(* IEC 61131-3 sources: TIA2AX/tests/V18/test_projects/expected/HW_2200330/ST30_PLC, 7 files *)

(* ---- HwIdentifiers.st ---- *)
TYPE
	HwIdentifiers : WORD
	(
		ST30_PLC_Profilschiene_0 :=	WORD#256,
		ST30_PLC :=	WORD#48,
		ST30_PLC_Card_reader_writer_1 :=	WORD#51,
		ST30_PLC_CPU_display_1 :=	WORD#54,
		ST30_PLC_OPC_UA_1 :=	WORD#117,
		ST30_PLC_DP_interface_1 :=	WORD#60,
		ST30_PLC_PROFINET_interface_1 :=	WORD#64,
		ST30_PLC_PROFINET_interface_1_Port_1 :=	WORD#65,
		ST30_PLC_PROFINET_interface_1_Port_2 :=	WORD#66,
		ST30_PLC_PROFINET_interface_2 :=	WORD#72,
		ST30_PLC_PROFINET_interface_2_Port_1 :=	WORD#73,
		ST30_Switch_SCALANCE_X_rack :=	WORD#436,
		ST30_Switch :=	WORD#437,
		ST30_Switch_ST30_Switch :=	WORD#438,
		ST30_Switch_SCALANCE_interface_1 :=	WORD#439,
		ST30_Switch_SCALANCE_interface_1_Port_1 :=	WORD#440,
		ST30_Switch_SCALANCE_interface_1_Port_2 :=	WORD#441,
		ST30_Switch_SCALANCE_interface_1_Port_3 :=	WORD#442,
		ST30_Switch_SCALANCE_interface_1_Port_4 :=	WORD#443,
		ST30_Switch_SCALANCE_interface_1_Port_5 :=	WORD#444,
		ST30_Switch_SCALANCE_interface_1_Port_6 :=	WORD#445,
		ST30_Switch_SCALANCE_interface_1_Port_7 :=	WORD#446,
		ST30_Switch_SCALANCE_interface_1_Port_8 :=	WORD#447,
		ST30_ET200SP_Rack_0 :=	WORD#276,
		ST30_ET200SP :=	WORD#277,
		ST30_ET200SP_ST30_ET200SP :=	WORD#258,
		ST30_ET200SP_PROFINET_interface :=	WORD#259,
		ST30_ET200SP_PROFINET_interface_Port_1 :=	WORD#260,
		ST30_ET200SP_PROFINET_interface_Port_2 :=	WORD#261,
		ST30_ET200SP_BA_2xRJ45 :=	WORD#260,
		ST30_ET200SP_CM_4xIO_Link_1 :=	WORD#262,
		ST30_ET200SP_CM_4xIO_Link_2 :=	WORD#263,
		ST30_ET200SP_DI_16x24VDC_ST_1 :=	WORD#264,
		ST30_ET200SP_DI_16x24VDC_ST_2 :=	WORD#265,
		ST30_ET200SP_DI_16x24VDC_ST_3 :=	WORD#266,
		ST30_ET200SP_DI_16x24VDC_ST_4 :=	WORD#267,
		ST30_ET200SP_DI_16x24VDC_ST_5 :=	WORD#268,
		ST30_ET200SP_DI_16x24VDC_ST_6 :=	WORD#269,
		ST30_ET200SP_DQ_16x24VDC_0_5A_ST_1 :=	WORD#270,
		ST30_ET200SP_DQ_16x24VDC_0_5A_ST_2 :=	WORD#271,
		ST30_ET200SP_DQ_16x24VDC_0_5A_ST_3 :=	WORD#272,
		ST30_ET200SP_DQ_16x24VDC_0_5A_ST_4 :=	WORD#273,
		ST30_ET200SP_Servermodul_1 :=	WORD#274,
		ST30_CPX_PN_IO_Interface :=	WORD#281,
		ST30_CPX_PN_IO_Interface_Port_1 :=	WORD#282,
		ST30_CPX_PN_IO_Interface_Port_2 :=	WORD#283,
		ST30_CPX_CPX :=	WORD#284,
		ST30_CPX_MPA1S_VMPA1_FB_EMS_8_8DO_1 :=	WORD#285,
		ST30_CPX_MPA1G_VMPA1_FB_EMG_8_8DO_1 :=	WORD#286,
		ST30_CPX_MPA1G_VMPA1_FB_EMG_8_8DO_2 :=	WORD#287,
		ST30_1_ACT350_Rack :=	WORD#289,
		ST30_1_ACT350 :=	WORD#290,
		ST30_1_ACT350_PROFINET :=	WORD#291,
		ST30_1_ACT350_PROFINET_Port_1 :=	WORD#292,
		ST30_1_ACT350_PROFINET_Port_2 :=	WORD#293,
		ST30_1_ACT350_DAP_2_Block_Parameter :=	WORD#294,
		ST30_1_ACT350_Measuring_Block_1 :=	WORD#295,
		ST30_1_ACT350_Measuring_Block_1_Parameter_Access_Point :=	WORD#296,
		ST30_1_ACT350_Measuring_Block_1_MB_Command_Value :=	WORD#297,
		ST30_1_ACT350_Measuring_Block_1_MB_Channel_Mask :=	WORD#298,
		ST30_1_ACT350_Measuring_Block_1_MB_Command :=	WORD#299,
		ST30_1_ACT350_Measuring_Block_1_MB_Measuring_Value :=	WORD#300,
		ST30_1_ACT350_Measuring_Block_1_MB_Device_Status :=	WORD#301,
		ST30_1_ACT350_Measuring_Block_1_MB_Response :=	WORD#302,
		ST30_1_ACT350_Status_Block_1 :=	WORD#303,
		ST30_1_ACT350_Status_Block_1_Parameter_Access_Point :=	WORD#304,
		ST30_1_ACT350_Status_Block_1_SB_Reserved_1 :=	WORD#305,
		ST30_1_ACT350_Status_Block_1_SB_Reserved_2 :=	WORD#306,
		ST30_1_ACT350_Status_Block_1_SB_Reserved_3 :=	WORD#307,
		ST30_1_ACT350_Status_Block_1_SB_Command :=	WORD#308,
		ST30_1_ACT350_Status_Block_1_SB_Status_Group_1 :=	WORD#309,
		ST30_1_ACT350_Status_Block_1_SB_Status_Group_2 :=	WORD#310,
		ST30_1_ACT350_Status_Block_1_SB_Status_Group_3 :=	WORD#311,
		ST30_1_ACT350_Status_Block_1_SB_Response :=	WORD#312,
		ST30_1_DM260_Rack :=	WORD#314,
		ST30_1_DM260 :=	WORD#315,
		ST30_1_DM260_Interface :=	WORD#316,
		ST30_1_DM260_Interface_Port_1 :=	WORD#317,
		ST30_1_DM260_DataMan_260 :=	WORD#318,
		ST30_1_DM260_Acquisition_Control_1 :=	WORD#319,
		ST30_1_DM260_Acquisition_Status_1 :=	WORD#320,
		ST30_1_DM260_Results_Control_1 :=	WORD#321,
		ST30_1_DM260_Results_Status_1 :=	WORD#322,
		ST30_1_DM260_Soft_Event_Control_1 :=	WORD#323,
		ST30_1_DM260_User_Data_64_bytes_1 :=	WORD#324,
		ST30_1_DM260_Result_Data_64_bytes_1 :=	WORD#325,
		ST30_1_CMMT_AS_X_PN_IO_Interface :=	WORD#329,
		ST30_1_CMMT_AS_X_PN_IO_Interface_Port_1 :=	WORD#330,
		ST30_1_CMMT_AS_X_PN_IO_Interface_Port_2 :=	WORD#331,
		ST30_1_CMMT_AS_X_CMMT_AS_V1 :=	WORD#332,
		ST30_1_CMMT_AS_X_DO_SERVO_1_Module_Access_Point :=	WORD#334,
		ST30_1_CMMT_AS_X_DO_SERVO_1_Siemens_telegram_111_PZD_12_12 :=	WORD#335,
		ST30_1_CMMT_AS_X_Siemens_telegram_111_PZD_12_12 :=	WORD#335,
		ST30_1_CMMT_AS_Y_PN_IO_Interface :=	WORD#339,
		ST30_1_CMMT_AS_Y_PN_IO_Interface_Port_1 :=	WORD#340,
		ST30_1_CMMT_AS_Y_PN_IO_Interface_Port_2 :=	WORD#341,
		ST30_1_CMMT_AS_Y_CMMT_AS_V1 :=	WORD#342,
		ST30_1_CMMT_AS_Y_DO_SERVO_1_Module_Access_Point :=	WORD#344,
		ST30_1_CMMT_AS_Y_DO_SERVO_1_Siemens_telegram_111_PZD_12_12 :=	WORD#345,
		ST30_1_CMMT_AS_Y_Siemens_telegram_111_PZD_12_12 :=	WORD#345,
		ST30_1_CMMT_AS_Z_PN_IO_Interface :=	WORD#349,
		ST30_1_CMMT_AS_Z_PN_IO_Interface_Port_1 :=	WORD#350,
		ST30_1_CMMT_AS_Z_PN_IO_Interface_Port_2 :=	WORD#351,
		ST30_1_CMMT_AS_Z_CMMT_AS_V1 :=	WORD#352,
		ST30_1_CMMT_AS_Z_DO_SERVO_1_Module_Access_Point :=	WORD#354,
		ST30_1_CMMT_AS_Z_DO_SERVO_1_Siemens_telegram_111_PZD_12_12 :=	WORD#355,
		ST30_1_CMMT_AS_Z_Siemens_telegram_111_PZD_12_12 :=	WORD#355,
		ST30_HMI_ConnectionBox_Connection_Box :=	WORD#357,
		ST30_HMI_ConnectionBox :=	WORD#358,
		ST30_HMI_ConnectionBox_ST30_HMI_ConnectionBox :=	WORD#359,
		ST30_HMI_ConnectionBox_SCALANCE_interface_1 :=	WORD#360,
		ST30_HMI_ConnectionBox_SCALANCE_interface_1_Port_1 :=	WORD#361,
		ST30_HMI_ConnectionBox_SCALANCE_interface_1_Port_2 :=	WORD#362,
		ST30_HMI_ConnectionBox_SCALANCE_interface_1_Port_3 :=	WORD#363,
		ST30_2_ACT350_Rack :=	WORD#365,
		ST30_2_ACT350 :=	WORD#366,
		ST30_2_ACT350_PROFINET :=	WORD#367,
		ST30_2_ACT350_PROFINET_Port_1 :=	WORD#368,
		ST30_2_ACT350_PROFINET_Port_2 :=	WORD#369,
		ST30_2_ACT350_DAP_2_Block_Parameter :=	WORD#370,
		ST30_2_ACT350_Measuring_Block_1 :=	WORD#371,
		ST30_2_ACT350_Measuring_Block_1_Parameter_Access_Point :=	WORD#372,
		ST30_2_ACT350_Measuring_Block_1_MB_Command_Value :=	WORD#373,
		ST30_2_ACT350_Measuring_Block_1_MB_Channel_Mask :=	WORD#374,
		ST30_2_ACT350_Measuring_Block_1_MB_Command :=	WORD#375,
		ST30_2_ACT350_Measuring_Block_1_MB_Measuring_Value :=	WORD#376,
		ST30_2_ACT350_Measuring_Block_1_MB_Device_Status :=	WORD#377,
		ST30_2_ACT350_Measuring_Block_1_MB_Response :=	WORD#378,
		ST30_2_ACT350_Status_Block_1 :=	WORD#379,
		ST30_2_ACT350_Status_Block_1_Parameter_Access_Point :=	WORD#380,
		ST30_2_ACT350_Status_Block_1_SB_Reserved_1 :=	WORD#381,
		ST30_2_ACT350_Status_Block_1_SB_Reserved_2 :=	WORD#382,
		ST30_2_ACT350_Status_Block_1_SB_Reserved_3 :=	WORD#383,
		ST30_2_ACT350_Status_Block_1_SB_Command :=	WORD#384,
		ST30_2_ACT350_Status_Block_1_SB_Status_Group_1 :=	WORD#385,
		ST30_2_ACT350_Status_Block_1_SB_Status_Group_2 :=	WORD#386,
		ST30_2_ACT350_Status_Block_1_SB_Status_Group_3 :=	WORD#387,
		ST30_2_ACT350_Status_Block_1_SB_Response :=	WORD#388,
		ST30_2_CMMT_AS_X_PN_IO_Interface :=	WORD#392,
		ST30_2_CMMT_AS_X_PN_IO_Interface_Port_1 :=	WORD#393,
		ST30_2_CMMT_AS_X_PN_IO_Interface_Port_2 :=	WORD#394,
		ST30_2_CMMT_AS_X_CMMT_AS_V1 :=	WORD#395,
		ST30_2_CMMT_AS_X_DO_SERVO_1_Module_Access_Point :=	WORD#397,
		ST30_2_CMMT_AS_X_DO_SERVO_1_Siemens_telegram_111_PZD_12_12 :=	WORD#398,
		ST30_2_CMMT_AS_X_Siemens_telegram_111_PZD_12_12 :=	WORD#398,
		ST30_2_CMMT_AS_Y_PN_IO_Interface :=	WORD#402,
		ST30_2_CMMT_AS_Y_PN_IO_Interface_Port_1 :=	WORD#403,
		ST30_2_CMMT_AS_Y_PN_IO_Interface_Port_2 :=	WORD#404,
		ST30_2_CMMT_AS_Y_CMMT_AS_V1 :=	WORD#405,
		ST30_2_CMMT_AS_Y_DO_SERVO_1_Module_Access_Point :=	WORD#407,
		ST30_2_CMMT_AS_Y_DO_SERVO_1_Siemens_telegram_111_PZD_12_12 :=	WORD#408,
		ST30_2_CMMT_AS_Y_Siemens_telegram_111_PZD_12_12 :=	WORD#408,
		ST30_2_CMMT_AS_Z_PN_IO_Interface :=	WORD#412,
		ST30_2_CMMT_AS_Z_PN_IO_Interface_Port_1 :=	WORD#413,
		ST30_2_CMMT_AS_Z_PN_IO_Interface_Port_2 :=	WORD#414,
		ST30_2_CMMT_AS_Z_CMMT_AS_V1 :=	WORD#415,
		ST30_2_CMMT_AS_Z_DO_SERVO_1_Module_Access_Point :=	WORD#417,
		ST30_2_CMMT_AS_Z_DO_SERVO_1_Siemens_telegram_111_PZD_12_12 :=	WORD#418,
		ST30_2_CMMT_AS_Z_Siemens_telegram_111_PZD_12_12 :=	WORD#418,
		ST30_2_DM260_Rack :=	WORD#420,
		ST30_2_DM260 :=	WORD#421,
		ST30_2_DM260_Interface :=	WORD#422,
		ST30_2_DM260_Interface_Port_1 :=	WORD#423,
		ST30_2_DM260_DataMan_260 :=	WORD#424,
		ST30_2_DM260_Acquisition_Control_1 :=	WORD#425,
		ST30_2_DM260_Acquisition_Status_1 :=	WORD#426,
		ST30_2_DM260_Results_Control_1 :=	WORD#427,
		ST30_2_DM260_Results_Status_1 :=	WORD#428,
		ST30_2_DM260_Soft_Event_Control_1 :=	WORD#429,
		ST30_2_DM260_User_Data_64_bytes_1 :=	WORD#430,
		ST30_2_DM260_Result_Data_64_bytes_1 :=	WORD#431,
		NONE:= WORD#0
	);
END_TYPE

(* ---- HwInputs.st ---- *)
TYPE
	HwInputs : STRUCT
		ST30_ET200SP_CM_4xIO_Link_1 AT %B100 : ARRAY[0..31] OF BYTE;
		ST30_ET200SP_CM_4xIO_Link_2 AT %B132 : ARRAY[0..31] OF BYTE;
		ST30_ET200SP_DI_16x24VDC_ST_1 AT %B0 : WORD;
		ST30_ET200SP_DI_16x24VDC_ST_2 AT %B2 : WORD;
		ST30_ET200SP_DI_16x24VDC_ST_3 AT %B4 : WORD;
		ST30_ET200SP_DI_16x24VDC_ST_4 AT %B6 : WORD;
		ST30_ET200SP_DI_16x24VDC_ST_5 AT %B8 : WORD;
		ST30_ET200SP_DI_16x24VDC_ST_6 AT %B10 : WORD;
		ST30_1_ACT350_Measuring_Block_1_MB_Measuring_Value AT %B1000 : DWORD;
		ST30_1_ACT350_Measuring_Block_1_MB_Device_Status AT %B1004 : WORD;
		ST30_1_ACT350_Measuring_Block_1_MB_Response AT %B1006 : WORD;
		ST30_1_ACT350_Status_Block_1_SB_Status_Group_1 AT %B1010 : WORD;
		ST30_1_ACT350_Status_Block_1_SB_Status_Group_2 AT %B1012 : WORD;
		ST30_1_ACT350_Status_Block_1_SB_Status_Group_3 AT %B1014 : WORD;
		ST30_1_ACT350_Status_Block_1_SB_Response AT %B1016 : WORD;
		ST30_1_DM260_Acquisition_Status_1 AT %B1500 : ARRAY[0..2] OF BYTE;
		ST30_1_DM260_Results_Status_1 AT %B1503 : BYTE;
		ST30_1_DM260_Soft_Event_Control_1 AT %B1504 : BYTE;
		ST30_1_DM260_Result_Data_64_bytes_1 AT %B1510 : ARRAY[0..71] OF BYTE;
		ST30_1_CMMT_AS_X_DO_SERVO_1_Siemens_telegram_111_PZD_12_12 AT %B1100 : ARRAY[0..23] OF BYTE;
		ST30_1_CMMT_AS_Y_DO_SERVO_1_Siemens_telegram_111_PZD_12_12 AT %B1200 : ARRAY[0..23] OF BYTE;
		ST30_1_CMMT_AS_Z_DO_SERVO_1_Siemens_telegram_111_PZD_12_12 AT %B1300 : ARRAY[0..23] OF BYTE;
		ST30_2_ACT350_Measuring_Block_1_MB_Measuring_Value AT %B2000 : DWORD;
		ST30_2_ACT350_Measuring_Block_1_MB_Device_Status AT %B2004 : WORD;
		ST30_2_ACT350_Measuring_Block_1_MB_Response AT %B2006 : WORD;
		ST30_2_ACT350_Status_Block_1_SB_Status_Group_1 AT %B2010 : WORD;
		ST30_2_ACT350_Status_Block_1_SB_Status_Group_2 AT %B2012 : WORD;
		ST30_2_ACT350_Status_Block_1_SB_Status_Group_3 AT %B2014 : WORD;
		ST30_2_ACT350_Status_Block_1_SB_Response AT %B2016 : WORD;
		ST30_2_CMMT_AS_X_DO_SERVO_1_Siemens_telegram_111_PZD_12_12 AT %B2100 : ARRAY[0..23] OF BYTE;
		ST30_2_CMMT_AS_Y_DO_SERVO_1_Siemens_telegram_111_PZD_12_12 AT %B2200 : ARRAY[0..23] OF BYTE;
		ST30_2_CMMT_AS_Z_DO_SERVO_1_Siemens_telegram_111_PZD_12_12 AT %B2300 : ARRAY[0..23] OF BYTE;
		ST30_2_DM260_Acquisition_Status_1 AT %B2500 : ARRAY[0..2] OF BYTE;
		ST30_2_DM260_Results_Status_1 AT %B2503 : BYTE;
		ST30_2_DM260_Soft_Event_Control_1 AT %B2504 : BYTE;
		ST30_2_DM260_Result_Data_64_bytes_1 AT %B2510 : ARRAY[0..71] OF BYTE;
	END_STRUCT;
END_TYPE

(* ---- HwOutputs.st ---- *)
TYPE
	HwOutputs : STRUCT
		ST30_ET200SP_CM_4xIO_Link_1 AT %B100 : ARRAY[0..31] OF BYTE;
		ST30_ET200SP_CM_4xIO_Link_2 AT %B132 : ARRAY[0..31] OF BYTE;
		ST30_ET200SP_DQ_16x24VDC_0_5A_ST_1 AT %B0 : WORD;
		ST30_ET200SP_DQ_16x24VDC_0_5A_ST_2 AT %B2 : WORD;
		ST30_ET200SP_DQ_16x24VDC_0_5A_ST_3 AT %B4 : WORD;
		ST30_ET200SP_DQ_16x24VDC_0_5A_ST_4 AT %B6 : WORD;
		ST30_CPX_MPA1S_VMPA1_FB_EMS_8_8DO_1 AT %B200 : BYTE;
		ST30_CPX_MPA1G_VMPA1_FB_EMG_8_8DO_1 AT %B201 : BYTE;
		ST30_CPX_MPA1G_VMPA1_FB_EMG_8_8DO_2 AT %B202 : BYTE;
		ST30_1_ACT350_Measuring_Block_1_MB_Command_Value AT %B1000 : DWORD;
		ST30_1_ACT350_Measuring_Block_1_MB_Channel_Mask AT %B1004 : WORD;
		ST30_1_ACT350_Measuring_Block_1_MB_Command AT %B1006 : WORD;
		ST30_1_ACT350_Status_Block_1_SB_Reserved_1 AT %B1010 : WORD;
		ST30_1_ACT350_Status_Block_1_SB_Reserved_2 AT %B1012 : WORD;
		ST30_1_ACT350_Status_Block_1_SB_Reserved_3 AT %B1014 : WORD;
		ST30_1_ACT350_Status_Block_1_SB_Command AT %B1016 : WORD;
		ST30_1_DM260_Acquisition_Control_1 AT %B1500 : BYTE;
		ST30_1_DM260_Results_Control_1 AT %B1503 : BYTE;
		ST30_1_DM260_Soft_Event_Control_1 AT %B1504 : BYTE;
		ST30_1_DM260_User_Data_64_bytes_1 AT %B1510 : ARRAY[0..67] OF BYTE;
		ST30_1_CMMT_AS_X_DO_SERVO_1_Siemens_telegram_111_PZD_12_12 AT %B1100 : ARRAY[0..23] OF BYTE;
		ST30_1_CMMT_AS_Y_DO_SERVO_1_Siemens_telegram_111_PZD_12_12 AT %B1200 : ARRAY[0..23] OF BYTE;
		ST30_1_CMMT_AS_Z_DO_SERVO_1_Siemens_telegram_111_PZD_12_12 AT %B1300 : ARRAY[0..23] OF BYTE;
		ST30_2_ACT350_Measuring_Block_1_MB_Command_Value AT %B2000 : DWORD;
		ST30_2_ACT350_Measuring_Block_1_MB_Channel_Mask AT %B2004 : WORD;
		ST30_2_ACT350_Measuring_Block_1_MB_Command AT %B2006 : WORD;
		ST30_2_ACT350_Status_Block_1_SB_Reserved_1 AT %B2010 : WORD;
		ST30_2_ACT350_Status_Block_1_SB_Reserved_2 AT %B2012 : WORD;
		ST30_2_ACT350_Status_Block_1_SB_Reserved_3 AT %B2014 : WORD;
		ST30_2_ACT350_Status_Block_1_SB_Command AT %B2016 : WORD;
		ST30_2_CMMT_AS_X_DO_SERVO_1_Siemens_telegram_111_PZD_12_12 AT %B2100 : ARRAY[0..23] OF BYTE;
		ST30_2_CMMT_AS_Y_DO_SERVO_1_Siemens_telegram_111_PZD_12_12 AT %B2200 : ARRAY[0..23] OF BYTE;
		ST30_2_CMMT_AS_Z_DO_SERVO_1_Siemens_telegram_111_PZD_12_12 AT %B2300 : ARRAY[0..23] OF BYTE;
		ST30_2_DM260_Acquisition_Control_1 AT %B2500 : BYTE;
		ST30_2_DM260_Results_Control_1 AT %B2503 : BYTE;
		ST30_2_DM260_Soft_Event_Control_1 AT %B2504 : BYTE;
		ST30_2_DM260_User_Data_64_bytes_1 AT %B2510 : ARRAY[0..67] OF BYTE;
	END_STRUCT;
END_TYPE

(* ---- PlcInputs.st ---- *)
TYPE
	PlcInputs : STRUCT
		ST30_ET200SP_CM_4xIO_Link_1 : ARRAY[0..31] OF BYTE;
		ST30_ET200SP_CM_4xIO_Link_2 : ARRAY[0..31] OF BYTE;
		ST30_ET200SP_DI_16x24VDC_ST_1 : WORD;
		ST30_ET200SP_DI_16x24VDC_ST_2 : WORD;
		ST30_ET200SP_DI_16x24VDC_ST_3 : WORD;
		ST30_ET200SP_DI_16x24VDC_ST_4 : WORD;
		ST30_ET200SP_DI_16x24VDC_ST_5 : WORD;
		ST30_ET200SP_DI_16x24VDC_ST_6 : WORD;
		ST30_1_ACT350_Measuring_Block_1_MB_Measuring_Value : DWORD;
		ST30_1_ACT350_Measuring_Block_1_MB_Device_Status : WORD;
		ST30_1_ACT350_Measuring_Block_1_MB_Response : WORD;
		ST30_1_ACT350_Status_Block_1_SB_Status_Group_1 : WORD;
		ST30_1_ACT350_Status_Block_1_SB_Status_Group_2 : WORD;
		ST30_1_ACT350_Status_Block_1_SB_Status_Group_3 : WORD;
		ST30_1_ACT350_Status_Block_1_SB_Response : WORD;
		ST30_1_DM260_Acquisition_Status_1 : ARRAY[0..2] OF BYTE;
		ST30_1_DM260_Results_Status_1 : BYTE;
		ST30_1_DM260_Soft_Event_Control_1 : BYTE;
		ST30_1_DM260_Result_Data_64_bytes_1 : ARRAY[0..71] OF BYTE;
		ST30_1_CMMT_AS_X_DO_SERVO_1_Siemens_telegram_111_PZD_12_12 : ARRAY[0..23] OF BYTE;
		ST30_1_CMMT_AS_Y_DO_SERVO_1_Siemens_telegram_111_PZD_12_12 : ARRAY[0..23] OF BYTE;
		ST30_1_CMMT_AS_Z_DO_SERVO_1_Siemens_telegram_111_PZD_12_12 : ARRAY[0..23] OF BYTE;
		ST30_2_ACT350_Measuring_Block_1_MB_Measuring_Value : DWORD;
		ST30_2_ACT350_Measuring_Block_1_MB_Device_Status : WORD;
		ST30_2_ACT350_Measuring_Block_1_MB_Response : WORD;
		ST30_2_ACT350_Status_Block_1_SB_Status_Group_1 : WORD;
		ST30_2_ACT350_Status_Block_1_SB_Status_Group_2 : WORD;
		ST30_2_ACT350_Status_Block_1_SB_Status_Group_3 : WORD;
		ST30_2_ACT350_Status_Block_1_SB_Response : WORD;
		ST30_2_CMMT_AS_X_DO_SERVO_1_Siemens_telegram_111_PZD_12_12 : ARRAY[0..23] OF BYTE;
		ST30_2_CMMT_AS_Y_DO_SERVO_1_Siemens_telegram_111_PZD_12_12 : ARRAY[0..23] OF BYTE;
		ST30_2_CMMT_AS_Z_DO_SERVO_1_Siemens_telegram_111_PZD_12_12 : ARRAY[0..23] OF BYTE;
		ST30_2_DM260_Acquisition_Status_1 : ARRAY[0..2] OF BYTE;
		ST30_2_DM260_Results_Status_1 : BYTE;
		ST30_2_DM260_Soft_Event_Control_1 : BYTE;
		ST30_2_DM260_Result_Data_64_bytes_1 : ARRAY[0..71] OF BYTE;
	END_STRUCT;
END_TYPE

(* ---- PlcOutputs.st ---- *)
TYPE
	PlcOutputs : STRUCT
		ST30_ET200SP_CM_4xIO_Link_1 : ARRAY[0..31] OF BYTE;
		ST30_ET200SP_CM_4xIO_Link_2 : ARRAY[0..31] OF BYTE;
		ST30_ET200SP_DQ_16x24VDC_0_5A_ST_1 : WORD;
		ST30_ET200SP_DQ_16x24VDC_0_5A_ST_2 : WORD;
		ST30_ET200SP_DQ_16x24VDC_0_5A_ST_3 : WORD;
		ST30_ET200SP_DQ_16x24VDC_0_5A_ST_4 : WORD;
		ST30_CPX_MPA1S_VMPA1_FB_EMS_8_8DO_1 : BYTE;
		ST30_CPX_MPA1G_VMPA1_FB_EMG_8_8DO_1 : BYTE;
		ST30_CPX_MPA1G_VMPA1_FB_EMG_8_8DO_2 : BYTE;
		ST30_1_ACT350_Measuring_Block_1_MB_Command_Value : DWORD;
		ST30_1_ACT350_Measuring_Block_1_MB_Channel_Mask : WORD;
		ST30_1_ACT350_Measuring_Block_1_MB_Command : WORD;
		ST30_1_ACT350_Status_Block_1_SB_Reserved_1 : WORD;
		ST30_1_ACT350_Status_Block_1_SB_Reserved_2 : WORD;
		ST30_1_ACT350_Status_Block_1_SB_Reserved_3 : WORD;
		ST30_1_ACT350_Status_Block_1_SB_Command : WORD;
		ST30_1_DM260_Acquisition_Control_1 : BYTE;
		ST30_1_DM260_Results_Control_1 : BYTE;
		ST30_1_DM260_Soft_Event_Control_1 : BYTE;
		ST30_1_DM260_User_Data_64_bytes_1 : ARRAY[0..67] OF BYTE;
		ST30_1_CMMT_AS_X_DO_SERVO_1_Siemens_telegram_111_PZD_12_12 : ARRAY[0..23] OF BYTE;
		ST30_1_CMMT_AS_Y_DO_SERVO_1_Siemens_telegram_111_PZD_12_12 : ARRAY[0..23] OF BYTE;
		ST30_1_CMMT_AS_Z_DO_SERVO_1_Siemens_telegram_111_PZD_12_12 : ARRAY[0..23] OF BYTE;
		ST30_2_ACT350_Measuring_Block_1_MB_Command_Value : DWORD;
		ST30_2_ACT350_Measuring_Block_1_MB_Channel_Mask : WORD;
		ST30_2_ACT350_Measuring_Block_1_MB_Command : WORD;
		ST30_2_ACT350_Status_Block_1_SB_Reserved_1 : WORD;
		ST30_2_ACT350_Status_Block_1_SB_Reserved_2 : WORD;
		ST30_2_ACT350_Status_Block_1_SB_Reserved_3 : WORD;
		ST30_2_ACT350_Status_Block_1_SB_Command : WORD;
		ST30_2_CMMT_AS_X_DO_SERVO_1_Siemens_telegram_111_PZD_12_12 : ARRAY[0..23] OF BYTE;
		ST30_2_CMMT_AS_Y_DO_SERVO_1_Siemens_telegram_111_PZD_12_12 : ARRAY[0..23] OF BYTE;
		ST30_2_CMMT_AS_Z_DO_SERVO_1_Siemens_telegram_111_PZD_12_12 : ARRAY[0..23] OF BYTE;
		ST30_2_DM260_Acquisition_Control_1 : BYTE;
		ST30_2_DM260_Results_Control_1 : BYTE;
		ST30_2_DM260_Soft_Event_Control_1 : BYTE;
		ST30_2_DM260_User_Data_64_bytes_1 : ARRAY[0..67] OF BYTE;
	END_STRUCT;
END_TYPE

(* ---- CopyInputs.st ---- *)
FUNCTION CopyInputs
	VAR_EXTERNAL
		HwInputs : HwInputs;
		PlcInputs : PlcInputs;
	END_VAR
	PlcInputs.ST30_ET200SP_CM_4xIO_Link_1[0] := HwInputs.ST30_ET200SP_CM_4xIO_Link_1[0];
	PlcInputs.ST30_ET200SP_CM_4xIO_Link_1[1] := HwInputs.ST30_ET200SP_CM_4xIO_Link_1[1];
	PlcInputs.ST30_ET200SP_CM_4xIO_Link_1[2] := HwInputs.ST30_ET200SP_CM_4xIO_Link_1[2];
	PlcInputs.ST30_ET200SP_CM_4xIO_Link_1[3] := HwInputs.ST30_ET200SP_CM_4xIO_Link_1[3];
	PlcInputs.ST30_ET200SP_CM_4xIO_Link_1[4] := HwInputs.ST30_ET200SP_CM_4xIO_Link_1[4];
	PlcInputs.ST30_ET200SP_CM_4xIO_Link_1[5] := HwInputs.ST30_ET200SP_CM_4xIO_Link_1[5];
	PlcInputs.ST30_ET200SP_CM_4xIO_Link_1[6] := HwInputs.ST30_ET200SP_CM_4xIO_Link_1[6];
	PlcInputs.ST30_ET200SP_CM_4xIO_Link_1[7] := HwInputs.ST30_ET200SP_CM_4xIO_Link_1[7];
	PlcInputs.ST30_ET200SP_CM_4xIO_Link_1[8] := HwInputs.ST30_ET200SP_CM_4xIO_Link_1[8];
	PlcInputs.ST30_ET200SP_CM_4xIO_Link_1[9] := HwInputs.ST30_ET200SP_CM_4xIO_Link_1[9];
	PlcInputs.ST30_ET200SP_CM_4xIO_Link_1[10] := HwInputs.ST30_ET200SP_CM_4xIO_Link_1[10];
	PlcInputs.ST30_ET200SP_CM_4xIO_Link_1[11] := HwInputs.ST30_ET200SP_CM_4xIO_Link_1[11];
	PlcInputs.ST30_ET200SP_CM_4xIO_Link_1[12] := HwInputs.ST30_ET200SP_CM_4xIO_Link_1[12];
	PlcInputs.ST30_ET200SP_CM_4xIO_Link_1[13] := HwInputs.ST30_ET200SP_CM_4xIO_Link_1[13];
	PlcInputs.ST30_ET200SP_CM_4xIO_Link_1[14] := HwInputs.ST30_ET200SP_CM_4xIO_Link_1[14];
	PlcInputs.ST30_ET200SP_CM_4xIO_Link_1[15] := HwInputs.ST30_ET200SP_CM_4xIO_Link_1[15];
	PlcInputs.ST30_ET200SP_CM_4xIO_Link_1[16] := HwInputs.ST30_ET200SP_CM_4xIO_Link_1[16];
	PlcInputs.ST30_ET200SP_CM_4xIO_Link_1[17] := HwInputs.ST30_ET200SP_CM_4xIO_Link_1[17];
	PlcInputs.ST30_ET200SP_CM_4xIO_Link_1[18] := HwInputs.ST30_ET200SP_CM_4xIO_Link_1[18];
	PlcInputs.ST30_ET200SP_CM_4xIO_Link_1[19] := HwInputs.ST30_ET200SP_CM_4xIO_Link_1[19];
	PlcInputs.ST30_ET200SP_CM_4xIO_Link_1[20] := HwInputs.ST30_ET200SP_CM_4xIO_Link_1[20];
	PlcInputs.ST30_ET200SP_CM_4xIO_Link_1[21] := HwInputs.ST30_ET200SP_CM_4xIO_Link_1[21];
	PlcInputs.ST30_ET200SP_CM_4xIO_Link_1[22] := HwInputs.ST30_ET200SP_CM_4xIO_Link_1[22];
	PlcInputs.ST30_ET200SP_CM_4xIO_Link_1[23] := HwInputs.ST30_ET200SP_CM_4xIO_Link_1[23];
	PlcInputs.ST30_ET200SP_CM_4xIO_Link_1[24] := HwInputs.ST30_ET200SP_CM_4xIO_Link_1[24];
	PlcInputs.ST30_ET200SP_CM_4xIO_Link_1[25] := HwInputs.ST30_ET200SP_CM_4xIO_Link_1[25];
	PlcInputs.ST30_ET200SP_CM_4xIO_Link_1[26] := HwInputs.ST30_ET200SP_CM_4xIO_Link_1[26];
	PlcInputs.ST30_ET200SP_CM_4xIO_Link_1[27] := HwInputs.ST30_ET200SP_CM_4xIO_Link_1[27];
	PlcInputs.ST30_ET200SP_CM_4xIO_Link_1[28] := HwInputs.ST30_ET200SP_CM_4xIO_Link_1[28];
	PlcInputs.ST30_ET200SP_CM_4xIO_Link_1[29] := HwInputs.ST30_ET200SP_CM_4xIO_Link_1[29];
	PlcInputs.ST30_ET200SP_CM_4xIO_Link_1[30] := HwInputs.ST30_ET200SP_CM_4xIO_Link_1[30];
	PlcInputs.ST30_ET200SP_CM_4xIO_Link_1[31] := HwInputs.ST30_ET200SP_CM_4xIO_Link_1[31];
	PlcInputs.ST30_ET200SP_CM_4xIO_Link_2[0] := HwInputs.ST30_ET200SP_CM_4xIO_Link_2[0];
	PlcInputs.ST30_ET200SP_CM_4xIO_Link_2[1] := HwInputs.ST30_ET200SP_CM_4xIO_Link_2[1];
	PlcInputs.ST30_ET200SP_CM_4xIO_Link_2[2] := HwInputs.ST30_ET200SP_CM_4xIO_Link_2[2];
	PlcInputs.ST30_ET200SP_CM_4xIO_Link_2[3] := HwInputs.ST30_ET200SP_CM_4xIO_Link_2[3];
	PlcInputs.ST30_ET200SP_CM_4xIO_Link_2[4] := HwInputs.ST30_ET200SP_CM_4xIO_Link_2[4];
	PlcInputs.ST30_ET200SP_CM_4xIO_Link_2[5] := HwInputs.ST30_ET200SP_CM_4xIO_Link_2[5];
	PlcInputs.ST30_ET200SP_CM_4xIO_Link_2[6] := HwInputs.ST30_ET200SP_CM_4xIO_Link_2[6];
	PlcInputs.ST30_ET200SP_CM_4xIO_Link_2[7] := HwInputs.ST30_ET200SP_CM_4xIO_Link_2[7];
	PlcInputs.ST30_ET200SP_CM_4xIO_Link_2[8] := HwInputs.ST30_ET200SP_CM_4xIO_Link_2[8];
	PlcInputs.ST30_ET200SP_CM_4xIO_Link_2[9] := HwInputs.ST30_ET200SP_CM_4xIO_Link_2[9];
	PlcInputs.ST30_ET200SP_CM_4xIO_Link_2[10] := HwInputs.ST30_ET200SP_CM_4xIO_Link_2[10];
	PlcInputs.ST30_ET200SP_CM_4xIO_Link_2[11] := HwInputs.ST30_ET200SP_CM_4xIO_Link_2[11];
	PlcInputs.ST30_ET200SP_CM_4xIO_Link_2[12] := HwInputs.ST30_ET200SP_CM_4xIO_Link_2[12];
	PlcInputs.ST30_ET200SP_CM_4xIO_Link_2[13] := HwInputs.ST30_ET200SP_CM_4xIO_Link_2[13];
	PlcInputs.ST30_ET200SP_CM_4xIO_Link_2[14] := HwInputs.ST30_ET200SP_CM_4xIO_Link_2[14];
	PlcInputs.ST30_ET200SP_CM_4xIO_Link_2[15] := HwInputs.ST30_ET200SP_CM_4xIO_Link_2[15];
	PlcInputs.ST30_ET200SP_CM_4xIO_Link_2[16] := HwInputs.ST30_ET200SP_CM_4xIO_Link_2[16];
	PlcInputs.ST30_ET200SP_CM_4xIO_Link_2[17] := HwInputs.ST30_ET200SP_CM_4xIO_Link_2[17];
	PlcInputs.ST30_ET200SP_CM_4xIO_Link_2[18] := HwInputs.ST30_ET200SP_CM_4xIO_Link_2[18];
	PlcInputs.ST30_ET200SP_CM_4xIO_Link_2[19] := HwInputs.ST30_ET200SP_CM_4xIO_Link_2[19];
	PlcInputs.ST30_ET200SP_CM_4xIO_Link_2[20] := HwInputs.ST30_ET200SP_CM_4xIO_Link_2[20];
	PlcInputs.ST30_ET200SP_CM_4xIO_Link_2[21] := HwInputs.ST30_ET200SP_CM_4xIO_Link_2[21];
	PlcInputs.ST30_ET200SP_CM_4xIO_Link_2[22] := HwInputs.ST30_ET200SP_CM_4xIO_Link_2[22];
	PlcInputs.ST30_ET200SP_CM_4xIO_Link_2[23] := HwInputs.ST30_ET200SP_CM_4xIO_Link_2[23];
	PlcInputs.ST30_ET200SP_CM_4xIO_Link_2[24] := HwInputs.ST30_ET200SP_CM_4xIO_Link_2[24];
	PlcInputs.ST30_ET200SP_CM_4xIO_Link_2[25] := HwInputs.ST30_ET200SP_CM_4xIO_Link_2[25];
	PlcInputs.ST30_ET200SP_CM_4xIO_Link_2[26] := HwInputs.ST30_ET200SP_CM_4xIO_Link_2[26];
	PlcInputs.ST30_ET200SP_CM_4xIO_Link_2[27] := HwInputs.ST30_ET200SP_CM_4xIO_Link_2[27];
	PlcInputs.ST30_ET200SP_CM_4xIO_Link_2[28] := HwInputs.ST30_ET200SP_CM_4xIO_Link_2[28];
	PlcInputs.ST30_ET200SP_CM_4xIO_Link_2[29] := HwInputs.ST30_ET200SP_CM_4xIO_Link_2[29];
	PlcInputs.ST30_ET200SP_CM_4xIO_Link_2[30] := HwInputs.ST30_ET200SP_CM_4xIO_Link_2[30];
	PlcInputs.ST30_ET200SP_CM_4xIO_Link_2[31] := HwInputs.ST30_ET200SP_CM_4xIO_Link_2[31];
	PlcInputs.ST30_ET200SP_DI_16x24VDC_ST_1 := HwInputs.ST30_ET200SP_DI_16x24VDC_ST_1;
	PlcInputs.ST30_ET200SP_DI_16x24VDC_ST_2 := HwInputs.ST30_ET200SP_DI_16x24VDC_ST_2;
	PlcInputs.ST30_ET200SP_DI_16x24VDC_ST_3 := HwInputs.ST30_ET200SP_DI_16x24VDC_ST_3;
	PlcInputs.ST30_ET200SP_DI_16x24VDC_ST_4 := HwInputs.ST30_ET200SP_DI_16x24VDC_ST_4;
	PlcInputs.ST30_ET200SP_DI_16x24VDC_ST_5 := HwInputs.ST30_ET200SP_DI_16x24VDC_ST_5;
	PlcInputs.ST30_ET200SP_DI_16x24VDC_ST_6 := HwInputs.ST30_ET200SP_DI_16x24VDC_ST_6;
	PlcInputs.ST30_1_ACT350_Measuring_Block_1_MB_Measuring_Value := HwInputs.ST30_1_ACT350_Measuring_Block_1_MB_Measuring_Value;
	PlcInputs.ST30_1_ACT350_Measuring_Block_1_MB_Device_Status := HwInputs.ST30_1_ACT350_Measuring_Block_1_MB_Device_Status;
	PlcInputs.ST30_1_ACT350_Measuring_Block_1_MB_Response := HwInputs.ST30_1_ACT350_Measuring_Block_1_MB_Response;
	PlcInputs.ST30_1_ACT350_Status_Block_1_SB_Status_Group_1 := HwInputs.ST30_1_ACT350_Status_Block_1_SB_Status_Group_1;
	PlcInputs.ST30_1_ACT350_Status_Block_1_SB_Status_Group_2 := HwInputs.ST30_1_ACT350_Status_Block_1_SB_Status_Group_2;
	PlcInputs.ST30_1_ACT350_Status_Block_1_SB_Status_Group_3 := HwInputs.ST30_1_ACT350_Status_Block_1_SB_Status_Group_3;
	PlcInputs.ST30_1_ACT350_Status_Block_1_SB_Response := HwInputs.ST30_1_ACT350_Status_Block_1_SB_Response;
	PlcInputs.ST30_1_DM260_Acquisition_Status_1[0] := HwInputs.ST30_1_DM260_Acquisition_Status_1[0];
	PlcInputs.ST30_1_DM260_Acquisition_Status_1[1] := HwInputs.ST30_1_DM260_Acquisition_Status_1[1];
	PlcInputs.ST30_1_DM260_Acquisition_Status_1[2] := HwInputs.ST30_1_DM260_Acquisition_Status_1[2];
	PlcInputs.ST30_1_DM260_Results_Status_1 := HwInputs.ST30_1_DM260_Results_Status_1;
	PlcInputs.ST30_1_DM260_Soft_Event_Control_1 := HwInputs.ST30_1_DM260_Soft_Event_Control_1;
	PlcInputs.ST30_1_DM260_Result_Data_64_bytes_1[0] := HwInputs.ST30_1_DM260_Result_Data_64_bytes_1[0];
	PlcInputs.ST30_1_DM260_Result_Data_64_bytes_1[1] := HwInputs.ST30_1_DM260_Result_Data_64_bytes_1[1];
	PlcInputs.ST30_1_DM260_Result_Data_64_bytes_1[2] := HwInputs.ST30_1_DM260_Result_Data_64_bytes_1[2];
	PlcInputs.ST30_1_DM260_Result_Data_64_bytes_1[3] := HwInputs.ST30_1_DM260_Result_Data_64_bytes_1[3];
	PlcInputs.ST30_1_DM260_Result_Data_64_bytes_1[4] := HwInputs.ST30_1_DM260_Result_Data_64_bytes_1[4];
	PlcInputs.ST30_1_DM260_Result_Data_64_bytes_1[5] := HwInputs.ST30_1_DM260_Result_Data_64_bytes_1[5];
	PlcInputs.ST30_1_DM260_Result_Data_64_bytes_1[6] := HwInputs.ST30_1_DM260_Result_Data_64_bytes_1[6];
	PlcInputs.ST30_1_DM260_Result_Data_64_bytes_1[7] := HwInputs.ST30_1_DM260_Result_Data_64_bytes_1[7];
	PlcInputs.ST30_1_DM260_Result_Data_64_bytes_1[8] := HwInputs.ST30_1_DM260_Result_Data_64_bytes_1[8];
	PlcInputs.ST30_1_DM260_Result_Data_64_bytes_1[9] := HwInputs.ST30_1_DM260_Result_Data_64_bytes_1[9];
	PlcInputs.ST30_1_DM260_Result_Data_64_bytes_1[10] := HwInputs.ST30_1_DM260_Result_Data_64_bytes_1[10];
	PlcInputs.ST30_1_DM260_Result_Data_64_bytes_1[11] := HwInputs.ST30_1_DM260_Result_Data_64_bytes_1[11];
	PlcInputs.ST30_1_DM260_Result_Data_64_bytes_1[12] := HwInputs.ST30_1_DM260_Result_Data_64_bytes_1[12];
	PlcInputs.ST30_1_DM260_Result_Data_64_bytes_1[13] := HwInputs.ST30_1_DM260_Result_Data_64_bytes_1[13];
	PlcInputs.ST30_1_DM260_Result_Data_64_bytes_1[14] := HwInputs.ST30_1_DM260_Result_Data_64_bytes_1[14];
	PlcInputs.ST30_1_DM260_Result_Data_64_bytes_1[15] := HwInputs.ST30_1_DM260_Result_Data_64_bytes_1[15];
	PlcInputs.ST30_1_DM260_Result_Data_64_bytes_1[16] := HwInputs.ST30_1_DM260_Result_Data_64_bytes_1[16];
	PlcInputs.ST30_1_DM260_Result_Data_64_bytes_1[17] := HwInputs.ST30_1_DM260_Result_Data_64_bytes_1[17];
	PlcInputs.ST30_1_DM260_Result_Data_64_bytes_1[18] := HwInputs.ST30_1_DM260_Result_Data_64_bytes_1[18];
	PlcInputs.ST30_1_DM260_Result_Data_64_bytes_1[19] := HwInputs.ST30_1_DM260_Result_Data_64_bytes_1[19];
	PlcInputs.ST30_1_DM260_Result_Data_64_bytes_1[20] := HwInputs.ST30_1_DM260_Result_Data_64_bytes_1[20];
	PlcInputs.ST30_1_DM260_Result_Data_64_bytes_1[21] := HwInputs.ST30_1_DM260_Result_Data_64_bytes_1[21];
	PlcInputs.ST30_1_DM260_Result_Data_64_bytes_1[22] := HwInputs.ST30_1_DM260_Result_Data_64_bytes_1[22];
	PlcInputs.ST30_1_DM260_Result_Data_64_bytes_1[23] := HwInputs.ST30_1_DM260_Result_Data_64_bytes_1[23];
	PlcInputs.ST30_1_DM260_Result_Data_64_bytes_1[24] := HwInputs.ST30_1_DM260_Result_Data_64_bytes_1[24];
	PlcInputs.ST30_1_DM260_Result_Data_64_bytes_1[25] := HwInputs.ST30_1_DM260_Result_Data_64_bytes_1[25];
	PlcInputs.ST30_1_DM260_Result_Data_64_bytes_1[26] := HwInputs.ST30_1_DM260_Result_Data_64_bytes_1[26];
	PlcInputs.ST30_1_DM260_Result_Data_64_bytes_1[27] := HwInputs.ST30_1_DM260_Result_Data_64_bytes_1[27];
	PlcInputs.ST30_1_DM260_Result_Data_64_bytes_1[28] := HwInputs.ST30_1_DM260_Result_Data_64_bytes_1[28];
	PlcInputs.ST30_1_DM260_Result_Data_64_bytes_1[29] := HwInputs.ST30_1_DM260_Result_Data_64_bytes_1[29];
	PlcInputs.ST30_1_DM260_Result_Data_64_bytes_1[30] := HwInputs.ST30_1_DM260_Result_Data_64_bytes_1[30];
	PlcInputs.ST30_1_DM260_Result_Data_64_bytes_1[31] := HwInputs.ST30_1_DM260_Result_Data_64_bytes_1[31];
	PlcInputs.ST30_1_DM260_Result_Data_64_bytes_1[32] := HwInputs.ST30_1_DM260_Result_Data_64_bytes_1[32];
	PlcInputs.ST30_1_DM260_Result_Data_64_bytes_1[33] := HwInputs.ST30_1_DM260_Result_Data_64_bytes_1[33];
	PlcInputs.ST30_1_DM260_Result_Data_64_bytes_1[34] := HwInputs.ST30_1_DM260_Result_Data_64_bytes_1[34];
	PlcInputs.ST30_1_DM260_Result_Data_64_bytes_1[35] := HwInputs.ST30_1_DM260_Result_Data_64_bytes_1[35];
	PlcInputs.ST30_1_DM260_Result_Data_64_bytes_1[36] := HwInputs.ST30_1_DM260_Result_Data_64_bytes_1[36];
	PlcInputs.ST30_1_DM260_Result_Data_64_bytes_1[37] := HwInputs.ST30_1_DM260_Result_Data_64_bytes_1[37];
	PlcInputs.ST30_1_DM260_Result_Data_64_bytes_1[38] := HwInputs.ST30_1_DM260_Result_Data_64_bytes_1[38];
	PlcInputs.ST30_1_DM260_Result_Data_64_bytes_1[39] := HwInputs.ST30_1_DM260_Result_Data_64_bytes_1[39];
	PlcInputs.ST30_1_DM260_Result_Data_64_bytes_1[40] := HwInputs.ST30_1_DM260_Result_Data_64_bytes_1[40];
	PlcInputs.ST30_1_DM260_Result_Data_64_bytes_1[41] := HwInputs.ST30_1_DM260_Result_Data_64_bytes_1[41];
	PlcInputs.ST30_1_DM260_Result_Data_64_bytes_1[42] := HwInputs.ST30_1_DM260_Result_Data_64_bytes_1[42];
	PlcInputs.ST30_1_DM260_Result_Data_64_bytes_1[43] := HwInputs.ST30_1_DM260_Result_Data_64_bytes_1[43];
	PlcInputs.ST30_1_DM260_Result_Data_64_bytes_1[44] := HwInputs.ST30_1_DM260_Result_Data_64_bytes_1[44];
	PlcInputs.ST30_1_DM260_Result_Data_64_bytes_1[45] := HwInputs.ST30_1_DM260_Result_Data_64_bytes_1[45];
	PlcInputs.ST30_1_DM260_Result_Data_64_bytes_1[46] := HwInputs.ST30_1_DM260_Result_Data_64_bytes_1[46];
	PlcInputs.ST30_1_DM260_Result_Data_64_bytes_1[47] := HwInputs.ST30_1_DM260_Result_Data_64_bytes_1[47];
	PlcInputs.ST30_1_DM260_Result_Data_64_bytes_1[48] := HwInputs.ST30_1_DM260_Result_Data_64_bytes_1[48];
	PlcInputs.ST30_1_DM260_Result_Data_64_bytes_1[49] := HwInputs.ST30_1_DM260_Result_Data_64_bytes_1[49];
	PlcInputs.ST30_1_DM260_Result_Data_64_bytes_1[50] := HwInputs.ST30_1_DM260_Result_Data_64_bytes_1[50];
	PlcInputs.ST30_1_DM260_Result_Data_64_bytes_1[51] := HwInputs.ST30_1_DM260_Result_Data_64_bytes_1[51];
	PlcInputs.ST30_1_DM260_Result_Data_64_bytes_1[52] := HwInputs.ST30_1_DM260_Result_Data_64_bytes_1[52];
	PlcInputs.ST30_1_DM260_Result_Data_64_bytes_1[53] := HwInputs.ST30_1_DM260_Result_Data_64_bytes_1[53];
	PlcInputs.ST30_1_DM260_Result_Data_64_bytes_1[54] := HwInputs.ST30_1_DM260_Result_Data_64_bytes_1[54];
	PlcInputs.ST30_1_DM260_Result_Data_64_bytes_1[55] := HwInputs.ST30_1_DM260_Result_Data_64_bytes_1[55];
	PlcInputs.ST30_1_DM260_Result_Data_64_bytes_1[56] := HwInputs.ST30_1_DM260_Result_Data_64_bytes_1[56];
	PlcInputs.ST30_1_DM260_Result_Data_64_bytes_1[57] := HwInputs.ST30_1_DM260_Result_Data_64_bytes_1[57];
	PlcInputs.ST30_1_DM260_Result_Data_64_bytes_1[58] := HwInputs.ST30_1_DM260_Result_Data_64_bytes_1[58];
	PlcInputs.ST30_1_DM260_Result_Data_64_bytes_1[59] := HwInputs.ST30_1_DM260_Result_Data_64_bytes_1[59];
	PlcInputs.ST30_1_DM260_Result_Data_64_bytes_1[60] := HwInputs.ST30_1_DM260_Result_Data_64_bytes_1[60];
	PlcInputs.ST30_1_DM260_Result_Data_64_bytes_1[61] := HwInputs.ST30_1_DM260_Result_Data_64_bytes_1[61];
	PlcInputs.ST30_1_DM260_Result_Data_64_bytes_1[62] := HwInputs.ST30_1_DM260_Result_Data_64_bytes_1[62];
	PlcInputs.ST30_1_DM260_Result_Data_64_bytes_1[63] := HwInputs.ST30_1_DM260_Result_Data_64_bytes_1[63];
	PlcInputs.ST30_1_DM260_Result_Data_64_bytes_1[64] := HwInputs.ST30_1_DM260_Result_Data_64_bytes_1[64];
	PlcInputs.ST30_1_DM260_Result_Data_64_bytes_1[65] := HwInputs.ST30_1_DM260_Result_Data_64_bytes_1[65];
	PlcInputs.ST30_1_DM260_Result_Data_64_bytes_1[66] := HwInputs.ST30_1_DM260_Result_Data_64_bytes_1[66];
	PlcInputs.ST30_1_DM260_Result_Data_64_bytes_1[67] := HwInputs.ST30_1_DM260_Result_Data_64_bytes_1[67];
	PlcInputs.ST30_1_DM260_Result_Data_64_bytes_1[68] := HwInputs.ST30_1_DM260_Result_Data_64_bytes_1[68];
	PlcInputs.ST30_1_DM260_Result_Data_64_bytes_1[69] := HwInputs.ST30_1_DM260_Result_Data_64_bytes_1[69];
	PlcInputs.ST30_1_DM260_Result_Data_64_bytes_1[70] := HwInputs.ST30_1_DM260_Result_Data_64_bytes_1[70];
	PlcInputs.ST30_1_DM260_Result_Data_64_bytes_1[71] := HwInputs.ST30_1_DM260_Result_Data_64_bytes_1[71];
	PlcInputs.ST30_1_CMMT_AS_X_DO_SERVO_1_Siemens_telegram_111_PZD_12_12[0] := HwInputs.ST30_1_CMMT_AS_X_DO_SERVO_1_Siemens_telegram_111_PZD_12_12[0];
	PlcInputs.ST30_1_CMMT_AS_X_DO_SERVO_1_Siemens_telegram_111_PZD_12_12[1] := HwInputs.ST30_1_CMMT_AS_X_DO_SERVO_1_Siemens_telegram_111_PZD_12_12[1];
	PlcInputs.ST30_1_CMMT_AS_X_DO_SERVO_1_Siemens_telegram_111_PZD_12_12[2] := HwInputs.ST30_1_CMMT_AS_X_DO_SERVO_1_Siemens_telegram_111_PZD_12_12[2];
	PlcInputs.ST30_1_CMMT_AS_X_DO_SERVO_1_Siemens_telegram_111_PZD_12_12[3] := HwInputs.ST30_1_CMMT_AS_X_DO_SERVO_1_Siemens_telegram_111_PZD_12_12[3];
	PlcInputs.ST30_1_CMMT_AS_X_DO_SERVO_1_Siemens_telegram_111_PZD_12_12[4] := HwInputs.ST30_1_CMMT_AS_X_DO_SERVO_1_Siemens_telegram_111_PZD_12_12[4];
	PlcInputs.ST30_1_CMMT_AS_X_DO_SERVO_1_Siemens_telegram_111_PZD_12_12[5] := HwInputs.ST30_1_CMMT_AS_X_DO_SERVO_1_Siemens_telegram_111_PZD_12_12[5];
	PlcInputs.ST30_1_CMMT_AS_X_DO_SERVO_1_Siemens_telegram_111_PZD_12_12[6] := HwInputs.ST30_1_CMMT_AS_X_DO_SERVO_1_Siemens_telegram_111_PZD_12_12[6];
	PlcInputs.ST30_1_CMMT_AS_X_DO_SERVO_1_Siemens_telegram_111_PZD_12_12[7] := HwInputs.ST30_1_CMMT_AS_X_DO_SERVO_1_Siemens_telegram_111_PZD_12_12[7];
	PlcInputs.ST30_1_CMMT_AS_X_DO_SERVO_1_Siemens_telegram_111_PZD_12_12[8] := HwInputs.ST30_1_CMMT_AS_X_DO_SERVO_1_Siemens_telegram_111_PZD_12_12[8];
	PlcInputs.ST30_1_CMMT_AS_X_DO_SERVO_1_Siemens_telegram_111_PZD_12_12[9] := HwInputs.ST30_1_CMMT_AS_X_DO_SERVO_1_Siemens_telegram_111_PZD_12_12[9];
	PlcInputs.ST30_1_CMMT_AS_X_DO_SERVO_1_Siemens_telegram_111_PZD_12_12[10] := HwInputs.ST30_1_CMMT_AS_X_DO_SERVO_1_Siemens_telegram_111_PZD_12_12[10];
	PlcInputs.ST30_1_CMMT_AS_X_DO_SERVO_1_Siemens_telegram_111_PZD_12_12[11] := HwInputs.ST30_1_CMMT_AS_X_DO_SERVO_1_Siemens_telegram_111_PZD_12_12[11];
	PlcInputs.ST30_1_CMMT_AS_X_DO_SERVO_1_Siemens_telegram_111_PZD_12_12[12] := HwInputs.ST30_1_CMMT_AS_X_DO_SERVO_1_Siemens_telegram_111_PZD_12_12[12];
	PlcInputs.ST30_1_CMMT_AS_X_DO_SERVO_1_Siemens_telegram_111_PZD_12_12[13] := HwInputs.ST30_1_CMMT_AS_X_DO_SERVO_1_Siemens_telegram_111_PZD_12_12[13];
	PlcInputs.ST30_1_CMMT_AS_X_DO_SERVO_1_Siemens_telegram_111_PZD_12_12[14] := HwInputs.ST30_1_CMMT_AS_X_DO_SERVO_1_Siemens_telegram_111_PZD_12_12[14];
	PlcInputs.ST30_1_CMMT_AS_X_DO_SERVO_1_Siemens_telegram_111_PZD_12_12[15] := HwInputs.ST30_1_CMMT_AS_X_DO_SERVO_1_Siemens_telegram_111_PZD_12_12[15];
	PlcInputs.ST30_1_CMMT_AS_X_DO_SERVO_1_Siemens_telegram_111_PZD_12_12[16] := HwInputs.ST30_1_CMMT_AS_X_DO_SERVO_1_Siemens_telegram_111_PZD_12_12[16];
	PlcInputs.ST30_1_CMMT_AS_X_DO_SERVO_1_Siemens_telegram_111_PZD_12_12[17] := HwInputs.ST30_1_CMMT_AS_X_DO_SERVO_1_Siemens_telegram_111_PZD_12_12[17];
	PlcInputs.ST30_1_CMMT_AS_X_DO_SERVO_1_Siemens_telegram_111_PZD_12_12[18] := HwInputs.ST30_1_CMMT_AS_X_DO_SERVO_1_Siemens_telegram_111_PZD_12_12[18];
	PlcInputs.ST30_1_CMMT_AS_X_DO_SERVO_1_Siemens_telegram_111_PZD_12_12[19] := HwInputs.ST30_1_CMMT_AS_X_DO_SERVO_1_Siemens_telegram_111_PZD_12_12[19];
	PlcInputs.ST30_1_CMMT_AS_X_DO_SERVO_1_Siemens_telegram_111_PZD_12_12[20] := HwInputs.ST30_1_CMMT_AS_X_DO_SERVO_1_Siemens_telegram_111_PZD_12_12[20];
	PlcInputs.ST30_1_CMMT_AS_X_DO_SERVO_1_Siemens_telegram_111_PZD_12_12[21] := HwInputs.ST30_1_CMMT_AS_X_DO_SERVO_1_Siemens_telegram_111_PZD_12_12[21];
	PlcInputs.ST30_1_CMMT_AS_X_DO_SERVO_1_Siemens_telegram_111_PZD_12_12[22] := HwInputs.ST30_1_CMMT_AS_X_DO_SERVO_1_Siemens_telegram_111_PZD_12_12[22];
	PlcInputs.ST30_1_CMMT_AS_X_DO_SERVO_1_Siemens_telegram_111_PZD_12_12[23] := HwInputs.ST30_1_CMMT_AS_X_DO_SERVO_1_Siemens_telegram_111_PZD_12_12[23];
	PlcInputs.ST30_1_CMMT_AS_Y_DO_SERVO_1_Siemens_telegram_111_PZD_12_12[0] := HwInputs.ST30_1_CMMT_AS_Y_DO_SERVO_1_Siemens_telegram_111_PZD_12_12[0];
	PlcInputs.ST30_1_CMMT_AS_Y_DO_SERVO_1_Siemens_telegram_111_PZD_12_12[1] := HwInputs.ST30_1_CMMT_AS_Y_DO_SERVO_1_Siemens_telegram_111_PZD_12_12[1];
	PlcInputs.ST30_1_CMMT_AS_Y_DO_SERVO_1_Siemens_telegram_111_PZD_12_12[2] := HwInputs.ST30_1_CMMT_AS_Y_DO_SERVO_1_Siemens_telegram_111_PZD_12_12[2];
	PlcInputs.ST30_1_CMMT_AS_Y_DO_SERVO_1_Siemens_telegram_111_PZD_12_12[3] := HwInputs.ST30_1_CMMT_AS_Y_DO_SERVO_1_Siemens_telegram_111_PZD_12_12[3];
	PlcInputs.ST30_1_CMMT_AS_Y_DO_SERVO_1_Siemens_telegram_111_PZD_12_12[4] := HwInputs.ST30_1_CMMT_AS_Y_DO_SERVO_1_Siemens_telegram_111_PZD_12_12[4];
	PlcInputs.ST30_1_CMMT_AS_Y_DO_SERVO_1_Siemens_telegram_111_PZD_12_12[5] := HwInputs.ST30_1_CMMT_AS_Y_DO_SERVO_1_Siemens_telegram_111_PZD_12_12[5];
	PlcInputs.ST30_1_CMMT_AS_Y_DO_SERVO_1_Siemens_telegram_111_PZD_12_12[6] := HwInputs.ST30_1_CMMT_AS_Y_DO_SERVO_1_Siemens_telegram_111_PZD_12_12[6];
	PlcInputs.ST30_1_CMMT_AS_Y_DO_SERVO_1_Siemens_telegram_111_PZD_12_12[7] := HwInputs.ST30_1_CMMT_AS_Y_DO_SERVO_1_Siemens_telegram_111_PZD_12_12[7];
	PlcInputs.ST30_1_CMMT_AS_Y_DO_SERVO_1_Siemens_telegram_111_PZD_12_12[8] := HwInputs.ST30_1_CMMT_AS_Y_DO_SERVO_1_Siemens_telegram_111_PZD_12_12[8];
	PlcInputs.ST30_1_CMMT_AS_Y_DO_SERVO_1_Siemens_telegram_111_PZD_12_12[9] := HwInputs.ST30_1_CMMT_AS_Y_DO_SERVO_1_Siemens_telegram_111_PZD_12_12[9];
	PlcInputs.ST30_1_CMMT_AS_Y_DO_SERVO_1_Siemens_telegram_111_PZD_12_12[10] := HwInputs.ST30_1_CMMT_AS_Y_DO_SERVO_1_Siemens_telegram_111_PZD_12_12[10];
	PlcInputs.ST30_1_CMMT_AS_Y_DO_SERVO_1_Siemens_telegram_111_PZD_12_12[11] := HwInputs.ST30_1_CMMT_AS_Y_DO_SERVO_1_Siemens_telegram_111_PZD_12_12[11];
	PlcInputs.ST30_1_CMMT_AS_Y_DO_SERVO_1_Siemens_telegram_111_PZD_12_12[12] := HwInputs.ST30_1_CMMT_AS_Y_DO_SERVO_1_Siemens_telegram_111_PZD_12_12[12];
	PlcInputs.ST30_1_CMMT_AS_Y_DO_SERVO_1_Siemens_telegram_111_PZD_12_12[13] := HwInputs.ST30_1_CMMT_AS_Y_DO_SERVO_1_Siemens_telegram_111_PZD_12_12[13];
	PlcInputs.ST30_1_CMMT_AS_Y_DO_SERVO_1_Siemens_telegram_111_PZD_12_12[14] := HwInputs.ST30_1_CMMT_AS_Y_DO_SERVO_1_Siemens_telegram_111_PZD_12_12[14];
	PlcInputs.ST30_1_CMMT_AS_Y_DO_SERVO_1_Siemens_telegram_111_PZD_12_12[15] := HwInputs.ST30_1_CMMT_AS_Y_DO_SERVO_1_Siemens_telegram_111_PZD_12_12[15];
	PlcInputs.ST30_1_CMMT_AS_Y_DO_SERVO_1_Siemens_telegram_111_PZD_12_12[16] := HwInputs.ST30_1_CMMT_AS_Y_DO_SERVO_1_Siemens_telegram_111_PZD_12_12[16];
	PlcInputs.ST30_1_CMMT_AS_Y_DO_SERVO_1_Siemens_telegram_111_PZD_12_12[17] := HwInputs.ST30_1_CMMT_AS_Y_DO_SERVO_1_Siemens_telegram_111_PZD_12_12[17];
	PlcInputs.ST30_1_CMMT_AS_Y_DO_SERVO_1_Siemens_telegram_111_PZD_12_12[18] := HwInputs.ST30_1_CMMT_AS_Y_DO_SERVO_1_Siemens_telegram_111_PZD_12_12[18];
	PlcInputs.ST30_1_CMMT_AS_Y_DO_SERVO_1_Siemens_telegram_111_PZD_12_12[19] := HwInputs.ST30_1_CMMT_AS_Y_DO_SERVO_1_Siemens_telegram_111_PZD_12_12[19];
	PlcInputs.ST30_1_CMMT_AS_Y_DO_SERVO_1_Siemens_telegram_111_PZD_12_12[20] := HwInputs.ST30_1_CMMT_AS_Y_DO_SERVO_1_Siemens_telegram_111_PZD_12_12[20];
	PlcInputs.ST30_1_CMMT_AS_Y_DO_SERVO_1_Siemens_telegram_111_PZD_12_12[21] := HwInputs.ST30_1_CMMT_AS_Y_DO_SERVO_1_Siemens_telegram_111_PZD_12_12[21];
	PlcInputs.ST30_1_CMMT_AS_Y_DO_SERVO_1_Siemens_telegram_111_PZD_12_12[22] := HwInputs.ST30_1_CMMT_AS_Y_DO_SERVO_1_Siemens_telegram_111_PZD_12_12[22];
	PlcInputs.ST30_1_CMMT_AS_Y_DO_SERVO_1_Siemens_telegram_111_PZD_12_12[23] := HwInputs.ST30_1_CMMT_AS_Y_DO_SERVO_1_Siemens_telegram_111_PZD_12_12[23];
	PlcInputs.ST30_1_CMMT_AS_Z_DO_SERVO_1_Siemens_telegram_111_PZD_12_12[0] := HwInputs.ST30_1_CMMT_AS_Z_DO_SERVO_1_Siemens_telegram_111_PZD_12_12[0];
	PlcInputs.ST30_1_CMMT_AS_Z_DO_SERVO_1_Siemens_telegram_111_PZD_12_12[1] := HwInputs.ST30_1_CMMT_AS_Z_DO_SERVO_1_Siemens_telegram_111_PZD_12_12[1];
	PlcInputs.ST30_1_CMMT_AS_Z_DO_SERVO_1_Siemens_telegram_111_PZD_12_12[2] := HwInputs.ST30_1_CMMT_AS_Z_DO_SERVO_1_Siemens_telegram_111_PZD_12_12[2];
	PlcInputs.ST30_1_CMMT_AS_Z_DO_SERVO_1_Siemens_telegram_111_PZD_12_12[3] := HwInputs.ST30_1_CMMT_AS_Z_DO_SERVO_1_Siemens_telegram_111_PZD_12_12[3];
	PlcInputs.ST30_1_CMMT_AS_Z_DO_SERVO_1_Siemens_telegram_111_PZD_12_12[4] := HwInputs.ST30_1_CMMT_AS_Z_DO_SERVO_1_Siemens_telegram_111_PZD_12_12[4];
	PlcInputs.ST30_1_CMMT_AS_Z_DO_SERVO_1_Siemens_telegram_111_PZD_12_12[5] := HwInputs.ST30_1_CMMT_AS_Z_DO_SERVO_1_Siemens_telegram_111_PZD_12_12[5];
	PlcInputs.ST30_1_CMMT_AS_Z_DO_SERVO_1_Siemens_telegram_111_PZD_12_12[6] := HwInputs.ST30_1_CMMT_AS_Z_DO_SERVO_1_Siemens_telegram_111_PZD_12_12[6];
	PlcInputs.ST30_1_CMMT_AS_Z_DO_SERVO_1_Siemens_telegram_111_PZD_12_12[7] := HwInputs.ST30_1_CMMT_AS_Z_DO_SERVO_1_Siemens_telegram_111_PZD_12_12[7];
	PlcInputs.ST30_1_CMMT_AS_Z_DO_SERVO_1_Siemens_telegram_111_PZD_12_12[8] := HwInputs.ST30_1_CMMT_AS_Z_DO_SERVO_1_Siemens_telegram_111_PZD_12_12[8];
	PlcInputs.ST30_1_CMMT_AS_Z_DO_SERVO_1_Siemens_telegram_111_PZD_12_12[9] := HwInputs.ST30_1_CMMT_AS_Z_DO_SERVO_1_Siemens_telegram_111_PZD_12_12[9];
	PlcInputs.ST30_1_CMMT_AS_Z_DO_SERVO_1_Siemens_telegram_111_PZD_12_12[10] := HwInputs.ST30_1_CMMT_AS_Z_DO_SERVO_1_Siemens_telegram_111_PZD_12_12[10];
	PlcInputs.ST30_1_CMMT_AS_Z_DO_SERVO_1_Siemens_telegram_111_PZD_12_12[11] := HwInputs.ST30_1_CMMT_AS_Z_DO_SERVO_1_Siemens_telegram_111_PZD_12_12[11];
	PlcInputs.ST30_1_CMMT_AS_Z_DO_SERVO_1_Siemens_telegram_111_PZD_12_12[12] := HwInputs.ST30_1_CMMT_AS_Z_DO_SERVO_1_Siemens_telegram_111_PZD_12_12[12];
	PlcInputs.ST30_1_CMMT_AS_Z_DO_SERVO_1_Siemens_telegram_111_PZD_12_12[13] := HwInputs.ST30_1_CMMT_AS_Z_DO_SERVO_1_Siemens_telegram_111_PZD_12_12[13];
	PlcInputs.ST30_1_CMMT_AS_Z_DO_SERVO_1_Siemens_telegram_111_PZD_12_12[14] := HwInputs.ST30_1_CMMT_AS_Z_DO_SERVO_1_Siemens_telegram_111_PZD_12_12[14];
	PlcInputs.ST30_1_CMMT_AS_Z_DO_SERVO_1_Siemens_telegram_111_PZD_12_12[15] := HwInputs.ST30_1_CMMT_AS_Z_DO_SERVO_1_Siemens_telegram_111_PZD_12_12[15];
	PlcInputs.ST30_1_CMMT_AS_Z_DO_SERVO_1_Siemens_telegram_111_PZD_12_12[16] := HwInputs.ST30_1_CMMT_AS_Z_DO_SERVO_1_Siemens_telegram_111_PZD_12_12[16];
	PlcInputs.ST30_1_CMMT_AS_Z_DO_SERVO_1_Siemens_telegram_111_PZD_12_12[17] := HwInputs.ST30_1_CMMT_AS_Z_DO_SERVO_1_Siemens_telegram_111_PZD_12_12[17];
	PlcInputs.ST30_1_CMMT_AS_Z_DO_SERVO_1_Siemens_telegram_111_PZD_12_12[18] := HwInputs.ST30_1_CMMT_AS_Z_DO_SERVO_1_Siemens_telegram_111_PZD_12_12[18];
	PlcInputs.ST30_1_CMMT_AS_Z_DO_SERVO_1_Siemens_telegram_111_PZD_12_12[19] := HwInputs.ST30_1_CMMT_AS_Z_DO_SERVO_1_Siemens_telegram_111_PZD_12_12[19];
	PlcInputs.ST30_1_CMMT_AS_Z_DO_SERVO_1_Siemens_telegram_111_PZD_12_12[20] := HwInputs.ST30_1_CMMT_AS_Z_DO_SERVO_1_Siemens_telegram_111_PZD_12_12[20];
	PlcInputs.ST30_1_CMMT_AS_Z_DO_SERVO_1_Siemens_telegram_111_PZD_12_12[21] := HwInputs.ST30_1_CMMT_AS_Z_DO_SERVO_1_Siemens_telegram_111_PZD_12_12[21];
	PlcInputs.ST30_1_CMMT_AS_Z_DO_SERVO_1_Siemens_telegram_111_PZD_12_12[22] := HwInputs.ST30_1_CMMT_AS_Z_DO_SERVO_1_Siemens_telegram_111_PZD_12_12[22];
	PlcInputs.ST30_1_CMMT_AS_Z_DO_SERVO_1_Siemens_telegram_111_PZD_12_12[23] := HwInputs.ST30_1_CMMT_AS_Z_DO_SERVO_1_Siemens_telegram_111_PZD_12_12[23];
	PlcInputs.ST30_2_ACT350_Measuring_Block_1_MB_Measuring_Value := HwInputs.ST30_2_ACT350_Measuring_Block_1_MB_Measuring_Value;
	PlcInputs.ST30_2_ACT350_Measuring_Block_1_MB_Device_Status := HwInputs.ST30_2_ACT350_Measuring_Block_1_MB_Device_Status;
	PlcInputs.ST30_2_ACT350_Measuring_Block_1_MB_Response := HwInputs.ST30_2_ACT350_Measuring_Block_1_MB_Response;
	PlcInputs.ST30_2_ACT350_Status_Block_1_SB_Status_Group_1 := HwInputs.ST30_2_ACT350_Status_Block_1_SB_Status_Group_1;
	PlcInputs.ST30_2_ACT350_Status_Block_1_SB_Status_Group_2 := HwInputs.ST30_2_ACT350_Status_Block_1_SB_Status_Group_2;
	PlcInputs.ST30_2_ACT350_Status_Block_1_SB_Status_Group_3 := HwInputs.ST30_2_ACT350_Status_Block_1_SB_Status_Group_3;
	PlcInputs.ST30_2_ACT350_Status_Block_1_SB_Response := HwInputs.ST30_2_ACT350_Status_Block_1_SB_Response;
	PlcInputs.ST30_2_CMMT_AS_X_DO_SERVO_1_Siemens_telegram_111_PZD_12_12[0] := HwInputs.ST30_2_CMMT_AS_X_DO_SERVO_1_Siemens_telegram_111_PZD_12_12[0];
	PlcInputs.ST30_2_CMMT_AS_X_DO_SERVO_1_Siemens_telegram_111_PZD_12_12[1] := HwInputs.ST30_2_CMMT_AS_X_DO_SERVO_1_Siemens_telegram_111_PZD_12_12[1];
	PlcInputs.ST30_2_CMMT_AS_X_DO_SERVO_1_Siemens_telegram_111_PZD_12_12[2] := HwInputs.ST30_2_CMMT_AS_X_DO_SERVO_1_Siemens_telegram_111_PZD_12_12[2];
	PlcInputs.ST30_2_CMMT_AS_X_DO_SERVO_1_Siemens_telegram_111_PZD_12_12[3] := HwInputs.ST30_2_CMMT_AS_X_DO_SERVO_1_Siemens_telegram_111_PZD_12_12[3];
	PlcInputs.ST30_2_CMMT_AS_X_DO_SERVO_1_Siemens_telegram_111_PZD_12_12[4] := HwInputs.ST30_2_CMMT_AS_X_DO_SERVO_1_Siemens_telegram_111_PZD_12_12[4];
	PlcInputs.ST30_2_CMMT_AS_X_DO_SERVO_1_Siemens_telegram_111_PZD_12_12[5] := HwInputs.ST30_2_CMMT_AS_X_DO_SERVO_1_Siemens_telegram_111_PZD_12_12[5];
	PlcInputs.ST30_2_CMMT_AS_X_DO_SERVO_1_Siemens_telegram_111_PZD_12_12[6] := HwInputs.ST30_2_CMMT_AS_X_DO_SERVO_1_Siemens_telegram_111_PZD_12_12[6];
	PlcInputs.ST30_2_CMMT_AS_X_DO_SERVO_1_Siemens_telegram_111_PZD_12_12[7] := HwInputs.ST30_2_CMMT_AS_X_DO_SERVO_1_Siemens_telegram_111_PZD_12_12[7];
	PlcInputs.ST30_2_CMMT_AS_X_DO_SERVO_1_Siemens_telegram_111_PZD_12_12[8] := HwInputs.ST30_2_CMMT_AS_X_DO_SERVO_1_Siemens_telegram_111_PZD_12_12[8];
	PlcInputs.ST30_2_CMMT_AS_X_DO_SERVO_1_Siemens_telegram_111_PZD_12_12[9] := HwInputs.ST30_2_CMMT_AS_X_DO_SERVO_1_Siemens_telegram_111_PZD_12_12[9];
	PlcInputs.ST30_2_CMMT_AS_X_DO_SERVO_1_Siemens_telegram_111_PZD_12_12[10] := HwInputs.ST30_2_CMMT_AS_X_DO_SERVO_1_Siemens_telegram_111_PZD_12_12[10];
	PlcInputs.ST30_2_CMMT_AS_X_DO_SERVO_1_Siemens_telegram_111_PZD_12_12[11] := HwInputs.ST30_2_CMMT_AS_X_DO_SERVO_1_Siemens_telegram_111_PZD_12_12[11];
	PlcInputs.ST30_2_CMMT_AS_X_DO_SERVO_1_Siemens_telegram_111_PZD_12_12[12] := HwInputs.ST30_2_CMMT_AS_X_DO_SERVO_1_Siemens_telegram_111_PZD_12_12[12];
	PlcInputs.ST30_2_CMMT_AS_X_DO_SERVO_1_Siemens_telegram_111_PZD_12_12[13] := HwInputs.ST30_2_CMMT_AS_X_DO_SERVO_1_Siemens_telegram_111_PZD_12_12[13];
	PlcInputs.ST30_2_CMMT_AS_X_DO_SERVO_1_Siemens_telegram_111_PZD_12_12[14] := HwInputs.ST30_2_CMMT_AS_X_DO_SERVO_1_Siemens_telegram_111_PZD_12_12[14];
	PlcInputs.ST30_2_CMMT_AS_X_DO_SERVO_1_Siemens_telegram_111_PZD_12_12[15] := HwInputs.ST30_2_CMMT_AS_X_DO_SERVO_1_Siemens_telegram_111_PZD_12_12[15];
	PlcInputs.ST30_2_CMMT_AS_X_DO_SERVO_1_Siemens_telegram_111_PZD_12_12[16] := HwInputs.ST30_2_CMMT_AS_X_DO_SERVO_1_Siemens_telegram_111_PZD_12_12[16];
	PlcInputs.ST30_2_CMMT_AS_X_DO_SERVO_1_Siemens_telegram_111_PZD_12_12[17] := HwInputs.ST30_2_CMMT_AS_X_DO_SERVO_1_Siemens_telegram_111_PZD_12_12[17];
	PlcInputs.ST30_2_CMMT_AS_X_DO_SERVO_1_Siemens_telegram_111_PZD_12_12[18] := HwInputs.ST30_2_CMMT_AS_X_DO_SERVO_1_Siemens_telegram_111_PZD_12_12[18];
	PlcInputs.ST30_2_CMMT_AS_X_DO_SERVO_1_Siemens_telegram_111_PZD_12_12[19] := HwInputs.ST30_2_CMMT_AS_X_DO_SERVO_1_Siemens_telegram_111_PZD_12_12[19];
	PlcInputs.ST30_2_CMMT_AS_X_DO_SERVO_1_Siemens_telegram_111_PZD_12_12[20] := HwInputs.ST30_2_CMMT_AS_X_DO_SERVO_1_Siemens_telegram_111_PZD_12_12[20];
	PlcInputs.ST30_2_CMMT_AS_X_DO_SERVO_1_Siemens_telegram_111_PZD_12_12[21] := HwInputs.ST30_2_CMMT_AS_X_DO_SERVO_1_Siemens_telegram_111_PZD_12_12[21];
	PlcInputs.ST30_2_CMMT_AS_X_DO_SERVO_1_Siemens_telegram_111_PZD_12_12[22] := HwInputs.ST30_2_CMMT_AS_X_DO_SERVO_1_Siemens_telegram_111_PZD_12_12[22];
	PlcInputs.ST30_2_CMMT_AS_X_DO_SERVO_1_Siemens_telegram_111_PZD_12_12[23] := HwInputs.ST30_2_CMMT_AS_X_DO_SERVO_1_Siemens_telegram_111_PZD_12_12[23];
	PlcInputs.ST30_2_CMMT_AS_Y_DO_SERVO_1_Siemens_telegram_111_PZD_12_12[0] := HwInputs.ST30_2_CMMT_AS_Y_DO_SERVO_1_Siemens_telegram_111_PZD_12_12[0];
	PlcInputs.ST30_2_CMMT_AS_Y_DO_SERVO_1_Siemens_telegram_111_PZD_12_12[1] := HwInputs.ST30_2_CMMT_AS_Y_DO_SERVO_1_Siemens_telegram_111_PZD_12_12[1];
	PlcInputs.ST30_2_CMMT_AS_Y_DO_SERVO_1_Siemens_telegram_111_PZD_12_12[2] := HwInputs.ST30_2_CMMT_AS_Y_DO_SERVO_1_Siemens_telegram_111_PZD_12_12[2];
	PlcInputs.ST30_2_CMMT_AS_Y_DO_SERVO_1_Siemens_telegram_111_PZD_12_12[3] := HwInputs.ST30_2_CMMT_AS_Y_DO_SERVO_1_Siemens_telegram_111_PZD_12_12[3];
	PlcInputs.ST30_2_CMMT_AS_Y_DO_SERVO_1_Siemens_telegram_111_PZD_12_12[4] := HwInputs.ST30_2_CMMT_AS_Y_DO_SERVO_1_Siemens_telegram_111_PZD_12_12[4];
	PlcInputs.ST30_2_CMMT_AS_Y_DO_SERVO_1_Siemens_telegram_111_PZD_12_12[5] := HwInputs.ST30_2_CMMT_AS_Y_DO_SERVO_1_Siemens_telegram_111_PZD_12_12[5];
	PlcInputs.ST30_2_CMMT_AS_Y_DO_SERVO_1_Siemens_telegram_111_PZD_12_12[6] := HwInputs.ST30_2_CMMT_AS_Y_DO_SERVO_1_Siemens_telegram_111_PZD_12_12[6];
	PlcInputs.ST30_2_CMMT_AS_Y_DO_SERVO_1_Siemens_telegram_111_PZD_12_12[7] := HwInputs.ST30_2_CMMT_AS_Y_DO_SERVO_1_Siemens_telegram_111_PZD_12_12[7];
	PlcInputs.ST30_2_CMMT_AS_Y_DO_SERVO_1_Siemens_telegram_111_PZD_12_12[8] := HwInputs.ST30_2_CMMT_AS_Y_DO_SERVO_1_Siemens_telegram_111_PZD_12_12[8];
	PlcInputs.ST30_2_CMMT_AS_Y_DO_SERVO_1_Siemens_telegram_111_PZD_12_12[9] := HwInputs.ST30_2_CMMT_AS_Y_DO_SERVO_1_Siemens_telegram_111_PZD_12_12[9];
	PlcInputs.ST30_2_CMMT_AS_Y_DO_SERVO_1_Siemens_telegram_111_PZD_12_12[10] := HwInputs.ST30_2_CMMT_AS_Y_DO_SERVO_1_Siemens_telegram_111_PZD_12_12[10];
	PlcInputs.ST30_2_CMMT_AS_Y_DO_SERVO_1_Siemens_telegram_111_PZD_12_12[11] := HwInputs.ST30_2_CMMT_AS_Y_DO_SERVO_1_Siemens_telegram_111_PZD_12_12[11];
	PlcInputs.ST30_2_CMMT_AS_Y_DO_SERVO_1_Siemens_telegram_111_PZD_12_12[12] := HwInputs.ST30_2_CMMT_AS_Y_DO_SERVO_1_Siemens_telegram_111_PZD_12_12[12];
	PlcInputs.ST30_2_CMMT_AS_Y_DO_SERVO_1_Siemens_telegram_111_PZD_12_12[13] := HwInputs.ST30_2_CMMT_AS_Y_DO_SERVO_1_Siemens_telegram_111_PZD_12_12[13];
	PlcInputs.ST30_2_CMMT_AS_Y_DO_SERVO_1_Siemens_telegram_111_PZD_12_12[14] := HwInputs.ST30_2_CMMT_AS_Y_DO_SERVO_1_Siemens_telegram_111_PZD_12_12[14];
	PlcInputs.ST30_2_CMMT_AS_Y_DO_SERVO_1_Siemens_telegram_111_PZD_12_12[15] := HwInputs.ST30_2_CMMT_AS_Y_DO_SERVO_1_Siemens_telegram_111_PZD_12_12[15];
	PlcInputs.ST30_2_CMMT_AS_Y_DO_SERVO_1_Siemens_telegram_111_PZD_12_12[16] := HwInputs.ST30_2_CMMT_AS_Y_DO_SERVO_1_Siemens_telegram_111_PZD_12_12[16];
	PlcInputs.ST30_2_CMMT_AS_Y_DO_SERVO_1_Siemens_telegram_111_PZD_12_12[17] := HwInputs.ST30_2_CMMT_AS_Y_DO_SERVO_1_Siemens_telegram_111_PZD_12_12[17];
	PlcInputs.ST30_2_CMMT_AS_Y_DO_SERVO_1_Siemens_telegram_111_PZD_12_12[18] := HwInputs.ST30_2_CMMT_AS_Y_DO_SERVO_1_Siemens_telegram_111_PZD_12_12[18];
	PlcInputs.ST30_2_CMMT_AS_Y_DO_SERVO_1_Siemens_telegram_111_PZD_12_12[19] := HwInputs.ST30_2_CMMT_AS_Y_DO_SERVO_1_Siemens_telegram_111_PZD_12_12[19];
	PlcInputs.ST30_2_CMMT_AS_Y_DO_SERVO_1_Siemens_telegram_111_PZD_12_12[20] := HwInputs.ST30_2_CMMT_AS_Y_DO_SERVO_1_Siemens_telegram_111_PZD_12_12[20];
	PlcInputs.ST30_2_CMMT_AS_Y_DO_SERVO_1_Siemens_telegram_111_PZD_12_12[21] := HwInputs.ST30_2_CMMT_AS_Y_DO_SERVO_1_Siemens_telegram_111_PZD_12_12[21];
	PlcInputs.ST30_2_CMMT_AS_Y_DO_SERVO_1_Siemens_telegram_111_PZD_12_12[22] := HwInputs.ST30_2_CMMT_AS_Y_DO_SERVO_1_Siemens_telegram_111_PZD_12_12[22];
	PlcInputs.ST30_2_CMMT_AS_Y_DO_SERVO_1_Siemens_telegram_111_PZD_12_12[23] := HwInputs.ST30_2_CMMT_AS_Y_DO_SERVO_1_Siemens_telegram_111_PZD_12_12[23];
	PlcInputs.ST30_2_CMMT_AS_Z_DO_SERVO_1_Siemens_telegram_111_PZD_12_12[0] := HwInputs.ST30_2_CMMT_AS_Z_DO_SERVO_1_Siemens_telegram_111_PZD_12_12[0];
	PlcInputs.ST30_2_CMMT_AS_Z_DO_SERVO_1_Siemens_telegram_111_PZD_12_12[1] := HwInputs.ST30_2_CMMT_AS_Z_DO_SERVO_1_Siemens_telegram_111_PZD_12_12[1];
	PlcInputs.ST30_2_CMMT_AS_Z_DO_SERVO_1_Siemens_telegram_111_PZD_12_12[2] := HwInputs.ST30_2_CMMT_AS_Z_DO_SERVO_1_Siemens_telegram_111_PZD_12_12[2];
	PlcInputs.ST30_2_CMMT_AS_Z_DO_SERVO_1_Siemens_telegram_111_PZD_12_12[3] := HwInputs.ST30_2_CMMT_AS_Z_DO_SERVO_1_Siemens_telegram_111_PZD_12_12[3];
	PlcInputs.ST30_2_CMMT_AS_Z_DO_SERVO_1_Siemens_telegram_111_PZD_12_12[4] := HwInputs.ST30_2_CMMT_AS_Z_DO_SERVO_1_Siemens_telegram_111_PZD_12_12[4];
	PlcInputs.ST30_2_CMMT_AS_Z_DO_SERVO_1_Siemens_telegram_111_PZD_12_12[5] := HwInputs.ST30_2_CMMT_AS_Z_DO_SERVO_1_Siemens_telegram_111_PZD_12_12[5];
	PlcInputs.ST30_2_CMMT_AS_Z_DO_SERVO_1_Siemens_telegram_111_PZD_12_12[6] := HwInputs.ST30_2_CMMT_AS_Z_DO_SERVO_1_Siemens_telegram_111_PZD_12_12[6];
	PlcInputs.ST30_2_CMMT_AS_Z_DO_SERVO_1_Siemens_telegram_111_PZD_12_12[7] := HwInputs.ST30_2_CMMT_AS_Z_DO_SERVO_1_Siemens_telegram_111_PZD_12_12[7];
	PlcInputs.ST30_2_CMMT_AS_Z_DO_SERVO_1_Siemens_telegram_111_PZD_12_12[8] := HwInputs.ST30_2_CMMT_AS_Z_DO_SERVO_1_Siemens_telegram_111_PZD_12_12[8];
	PlcInputs.ST30_2_CMMT_AS_Z_DO_SERVO_1_Siemens_telegram_111_PZD_12_12[9] := HwInputs.ST30_2_CMMT_AS_Z_DO_SERVO_1_Siemens_telegram_111_PZD_12_12[9];
	PlcInputs.ST30_2_CMMT_AS_Z_DO_SERVO_1_Siemens_telegram_111_PZD_12_12[10] := HwInputs.ST30_2_CMMT_AS_Z_DO_SERVO_1_Siemens_telegram_111_PZD_12_12[10];
	PlcInputs.ST30_2_CMMT_AS_Z_DO_SERVO_1_Siemens_telegram_111_PZD_12_12[11] := HwInputs.ST30_2_CMMT_AS_Z_DO_SERVO_1_Siemens_telegram_111_PZD_12_12[11];
	PlcInputs.ST30_2_CMMT_AS_Z_DO_SERVO_1_Siemens_telegram_111_PZD_12_12[12] := HwInputs.ST30_2_CMMT_AS_Z_DO_SERVO_1_Siemens_telegram_111_PZD_12_12[12];
	PlcInputs.ST30_2_CMMT_AS_Z_DO_SERVO_1_Siemens_telegram_111_PZD_12_12[13] := HwInputs.ST30_2_CMMT_AS_Z_DO_SERVO_1_Siemens_telegram_111_PZD_12_12[13];
	PlcInputs.ST30_2_CMMT_AS_Z_DO_SERVO_1_Siemens_telegram_111_PZD_12_12[14] := HwInputs.ST30_2_CMMT_AS_Z_DO_SERVO_1_Siemens_telegram_111_PZD_12_12[14];
	PlcInputs.ST30_2_CMMT_AS_Z_DO_SERVO_1_Siemens_telegram_111_PZD_12_12[15] := HwInputs.ST30_2_CMMT_AS_Z_DO_SERVO_1_Siemens_telegram_111_PZD_12_12[15];
	PlcInputs.ST30_2_CMMT_AS_Z_DO_SERVO_1_Siemens_telegram_111_PZD_12_12[16] := HwInputs.ST30_2_CMMT_AS_Z_DO_SERVO_1_Siemens_telegram_111_PZD_12_12[16];
	PlcInputs.ST30_2_CMMT_AS_Z_DO_SERVO_1_Siemens_telegram_111_PZD_12_12[17] := HwInputs.ST30_2_CMMT_AS_Z_DO_SERVO_1_Siemens_telegram_111_PZD_12_12[17];
	PlcInputs.ST30_2_CMMT_AS_Z_DO_SERVO_1_Siemens_telegram_111_PZD_12_12[18] := HwInputs.ST30_2_CMMT_AS_Z_DO_SERVO_1_Siemens_telegram_111_PZD_12_12[18];
	PlcInputs.ST30_2_CMMT_AS_Z_DO_SERVO_1_Siemens_telegram_111_PZD_12_12[19] := HwInputs.ST30_2_CMMT_AS_Z_DO_SERVO_1_Siemens_telegram_111_PZD_12_12[19];
	PlcInputs.ST30_2_CMMT_AS_Z_DO_SERVO_1_Siemens_telegram_111_PZD_12_12[20] := HwInputs.ST30_2_CMMT_AS_Z_DO_SERVO_1_Siemens_telegram_111_PZD_12_12[20];
	PlcInputs.ST30_2_CMMT_AS_Z_DO_SERVO_1_Siemens_telegram_111_PZD_12_12[21] := HwInputs.ST30_2_CMMT_AS_Z_DO_SERVO_1_Siemens_telegram_111_PZD_12_12[21];
	PlcInputs.ST30_2_CMMT_AS_Z_DO_SERVO_1_Siemens_telegram_111_PZD_12_12[22] := HwInputs.ST30_2_CMMT_AS_Z_DO_SERVO_1_Siemens_telegram_111_PZD_12_12[22];
	PlcInputs.ST30_2_CMMT_AS_Z_DO_SERVO_1_Siemens_telegram_111_PZD_12_12[23] := HwInputs.ST30_2_CMMT_AS_Z_DO_SERVO_1_Siemens_telegram_111_PZD_12_12[23];
	PlcInputs.ST30_2_DM260_Acquisition_Status_1[0] := HwInputs.ST30_2_DM260_Acquisition_Status_1[0];
	PlcInputs.ST30_2_DM260_Acquisition_Status_1[1] := HwInputs.ST30_2_DM260_Acquisition_Status_1[1];
	PlcInputs.ST30_2_DM260_Acquisition_Status_1[2] := HwInputs.ST30_2_DM260_Acquisition_Status_1[2];
	PlcInputs.ST30_2_DM260_Results_Status_1 := HwInputs.ST30_2_DM260_Results_Status_1;
	PlcInputs.ST30_2_DM260_Soft_Event_Control_1 := HwInputs.ST30_2_DM260_Soft_Event_Control_1;
	PlcInputs.ST30_2_DM260_Result_Data_64_bytes_1[0] := HwInputs.ST30_2_DM260_Result_Data_64_bytes_1[0];
	PlcInputs.ST30_2_DM260_Result_Data_64_bytes_1[1] := HwInputs.ST30_2_DM260_Result_Data_64_bytes_1[1];
	PlcInputs.ST30_2_DM260_Result_Data_64_bytes_1[2] := HwInputs.ST30_2_DM260_Result_Data_64_bytes_1[2];
	PlcInputs.ST30_2_DM260_Result_Data_64_bytes_1[3] := HwInputs.ST30_2_DM260_Result_Data_64_bytes_1[3];
	PlcInputs.ST30_2_DM260_Result_Data_64_bytes_1[4] := HwInputs.ST30_2_DM260_Result_Data_64_bytes_1[4];
	PlcInputs.ST30_2_DM260_Result_Data_64_bytes_1[5] := HwInputs.ST30_2_DM260_Result_Data_64_bytes_1[5];
	PlcInputs.ST30_2_DM260_Result_Data_64_bytes_1[6] := HwInputs.ST30_2_DM260_Result_Data_64_bytes_1[6];
	PlcInputs.ST30_2_DM260_Result_Data_64_bytes_1[7] := HwInputs.ST30_2_DM260_Result_Data_64_bytes_1[7];
	PlcInputs.ST30_2_DM260_Result_Data_64_bytes_1[8] := HwInputs.ST30_2_DM260_Result_Data_64_bytes_1[8];
	PlcInputs.ST30_2_DM260_Result_Data_64_bytes_1[9] := HwInputs.ST30_2_DM260_Result_Data_64_bytes_1[9];
	PlcInputs.ST30_2_DM260_Result_Data_64_bytes_1[10] := HwInputs.ST30_2_DM260_Result_Data_64_bytes_1[10];
	PlcInputs.ST30_2_DM260_Result_Data_64_bytes_1[11] := HwInputs.ST30_2_DM260_Result_Data_64_bytes_1[11];
	PlcInputs.ST30_2_DM260_Result_Data_64_bytes_1[12] := HwInputs.ST30_2_DM260_Result_Data_64_bytes_1[12];
	PlcInputs.ST30_2_DM260_Result_Data_64_bytes_1[13] := HwInputs.ST30_2_DM260_Result_Data_64_bytes_1[13];
	PlcInputs.ST30_2_DM260_Result_Data_64_bytes_1[14] := HwInputs.ST30_2_DM260_Result_Data_64_bytes_1[14];
	PlcInputs.ST30_2_DM260_Result_Data_64_bytes_1[15] := HwInputs.ST30_2_DM260_Result_Data_64_bytes_1[15];
	PlcInputs.ST30_2_DM260_Result_Data_64_bytes_1[16] := HwInputs.ST30_2_DM260_Result_Data_64_bytes_1[16];
	PlcInputs.ST30_2_DM260_Result_Data_64_bytes_1[17] := HwInputs.ST30_2_DM260_Result_Data_64_bytes_1[17];
	PlcInputs.ST30_2_DM260_Result_Data_64_bytes_1[18] := HwInputs.ST30_2_DM260_Result_Data_64_bytes_1[18];
	PlcInputs.ST30_2_DM260_Result_Data_64_bytes_1[19] := HwInputs.ST30_2_DM260_Result_Data_64_bytes_1[19];
	PlcInputs.ST30_2_DM260_Result_Data_64_bytes_1[20] := HwInputs.ST30_2_DM260_Result_Data_64_bytes_1[20];
	PlcInputs.ST30_2_DM260_Result_Data_64_bytes_1[21] := HwInputs.ST30_2_DM260_Result_Data_64_bytes_1[21];
	PlcInputs.ST30_2_DM260_Result_Data_64_bytes_1[22] := HwInputs.ST30_2_DM260_Result_Data_64_bytes_1[22];
	PlcInputs.ST30_2_DM260_Result_Data_64_bytes_1[23] := HwInputs.ST30_2_DM260_Result_Data_64_bytes_1[23];
	PlcInputs.ST30_2_DM260_Result_Data_64_bytes_1[24] := HwInputs.ST30_2_DM260_Result_Data_64_bytes_1[24];
	PlcInputs.ST30_2_DM260_Result_Data_64_bytes_1[25] := HwInputs.ST30_2_DM260_Result_Data_64_bytes_1[25];
	PlcInputs.ST30_2_DM260_Result_Data_64_bytes_1[26] := HwInputs.ST30_2_DM260_Result_Data_64_bytes_1[26];
	PlcInputs.ST30_2_DM260_Result_Data_64_bytes_1[27] := HwInputs.ST30_2_DM260_Result_Data_64_bytes_1[27];
	PlcInputs.ST30_2_DM260_Result_Data_64_bytes_1[28] := HwInputs.ST30_2_DM260_Result_Data_64_bytes_1[28];
	PlcInputs.ST30_2_DM260_Result_Data_64_bytes_1[29] := HwInputs.ST30_2_DM260_Result_Data_64_bytes_1[29];
	PlcInputs.ST30_2_DM260_Result_Data_64_bytes_1[30] := HwInputs.ST30_2_DM260_Result_Data_64_bytes_1[30];
	PlcInputs.ST30_2_DM260_Result_Data_64_bytes_1[31] := HwInputs.ST30_2_DM260_Result_Data_64_bytes_1[31];
	PlcInputs.ST30_2_DM260_Result_Data_64_bytes_1[32] := HwInputs.ST30_2_DM260_Result_Data_64_bytes_1[32];
	PlcInputs.ST30_2_DM260_Result_Data_64_bytes_1[33] := HwInputs.ST30_2_DM260_Result_Data_64_bytes_1[33];
	PlcInputs.ST30_2_DM260_Result_Data_64_bytes_1[34] := HwInputs.ST30_2_DM260_Result_Data_64_bytes_1[34];
	PlcInputs.ST30_2_DM260_Result_Data_64_bytes_1[35] := HwInputs.ST30_2_DM260_Result_Data_64_bytes_1[35];
	PlcInputs.ST30_2_DM260_Result_Data_64_bytes_1[36] := HwInputs.ST30_2_DM260_Result_Data_64_bytes_1[36];
	PlcInputs.ST30_2_DM260_Result_Data_64_bytes_1[37] := HwInputs.ST30_2_DM260_Result_Data_64_bytes_1[37];
	PlcInputs.ST30_2_DM260_Result_Data_64_bytes_1[38] := HwInputs.ST30_2_DM260_Result_Data_64_bytes_1[38];
	PlcInputs.ST30_2_DM260_Result_Data_64_bytes_1[39] := HwInputs.ST30_2_DM260_Result_Data_64_bytes_1[39];
	PlcInputs.ST30_2_DM260_Result_Data_64_bytes_1[40] := HwInputs.ST30_2_DM260_Result_Data_64_bytes_1[40];
	PlcInputs.ST30_2_DM260_Result_Data_64_bytes_1[41] := HwInputs.ST30_2_DM260_Result_Data_64_bytes_1[41];
	PlcInputs.ST30_2_DM260_Result_Data_64_bytes_1[42] := HwInputs.ST30_2_DM260_Result_Data_64_bytes_1[42];
	PlcInputs.ST30_2_DM260_Result_Data_64_bytes_1[43] := HwInputs.ST30_2_DM260_Result_Data_64_bytes_1[43];
	PlcInputs.ST30_2_DM260_Result_Data_64_bytes_1[44] := HwInputs.ST30_2_DM260_Result_Data_64_bytes_1[44];
	PlcInputs.ST30_2_DM260_Result_Data_64_bytes_1[45] := HwInputs.ST30_2_DM260_Result_Data_64_bytes_1[45];
	PlcInputs.ST30_2_DM260_Result_Data_64_bytes_1[46] := HwInputs.ST30_2_DM260_Result_Data_64_bytes_1[46];
	PlcInputs.ST30_2_DM260_Result_Data_64_bytes_1[47] := HwInputs.ST30_2_DM260_Result_Data_64_bytes_1[47];
	PlcInputs.ST30_2_DM260_Result_Data_64_bytes_1[48] := HwInputs.ST30_2_DM260_Result_Data_64_bytes_1[48];
	PlcInputs.ST30_2_DM260_Result_Data_64_bytes_1[49] := HwInputs.ST30_2_DM260_Result_Data_64_bytes_1[49];
	PlcInputs.ST30_2_DM260_Result_Data_64_bytes_1[50] := HwInputs.ST30_2_DM260_Result_Data_64_bytes_1[50];
	PlcInputs.ST30_2_DM260_Result_Data_64_bytes_1[51] := HwInputs.ST30_2_DM260_Result_Data_64_bytes_1[51];
	PlcInputs.ST30_2_DM260_Result_Data_64_bytes_1[52] := HwInputs.ST30_2_DM260_Result_Data_64_bytes_1[52];
	PlcInputs.ST30_2_DM260_Result_Data_64_bytes_1[53] := HwInputs.ST30_2_DM260_Result_Data_64_bytes_1[53];
	PlcInputs.ST30_2_DM260_Result_Data_64_bytes_1[54] := HwInputs.ST30_2_DM260_Result_Data_64_bytes_1[54];
	PlcInputs.ST30_2_DM260_Result_Data_64_bytes_1[55] := HwInputs.ST30_2_DM260_Result_Data_64_bytes_1[55];
	PlcInputs.ST30_2_DM260_Result_Data_64_bytes_1[56] := HwInputs.ST30_2_DM260_Result_Data_64_bytes_1[56];
	PlcInputs.ST30_2_DM260_Result_Data_64_bytes_1[57] := HwInputs.ST30_2_DM260_Result_Data_64_bytes_1[57];
	PlcInputs.ST30_2_DM260_Result_Data_64_bytes_1[58] := HwInputs.ST30_2_DM260_Result_Data_64_bytes_1[58];
	PlcInputs.ST30_2_DM260_Result_Data_64_bytes_1[59] := HwInputs.ST30_2_DM260_Result_Data_64_bytes_1[59];
	PlcInputs.ST30_2_DM260_Result_Data_64_bytes_1[60] := HwInputs.ST30_2_DM260_Result_Data_64_bytes_1[60];
	PlcInputs.ST30_2_DM260_Result_Data_64_bytes_1[61] := HwInputs.ST30_2_DM260_Result_Data_64_bytes_1[61];
	PlcInputs.ST30_2_DM260_Result_Data_64_bytes_1[62] := HwInputs.ST30_2_DM260_Result_Data_64_bytes_1[62];
	PlcInputs.ST30_2_DM260_Result_Data_64_bytes_1[63] := HwInputs.ST30_2_DM260_Result_Data_64_bytes_1[63];
	PlcInputs.ST30_2_DM260_Result_Data_64_bytes_1[64] := HwInputs.ST30_2_DM260_Result_Data_64_bytes_1[64];
	PlcInputs.ST30_2_DM260_Result_Data_64_bytes_1[65] := HwInputs.ST30_2_DM260_Result_Data_64_bytes_1[65];
	PlcInputs.ST30_2_DM260_Result_Data_64_bytes_1[66] := HwInputs.ST30_2_DM260_Result_Data_64_bytes_1[66];
	PlcInputs.ST30_2_DM260_Result_Data_64_bytes_1[67] := HwInputs.ST30_2_DM260_Result_Data_64_bytes_1[67];
	PlcInputs.ST30_2_DM260_Result_Data_64_bytes_1[68] := HwInputs.ST30_2_DM260_Result_Data_64_bytes_1[68];
	PlcInputs.ST30_2_DM260_Result_Data_64_bytes_1[69] := HwInputs.ST30_2_DM260_Result_Data_64_bytes_1[69];
	PlcInputs.ST30_2_DM260_Result_Data_64_bytes_1[70] := HwInputs.ST30_2_DM260_Result_Data_64_bytes_1[70];
	PlcInputs.ST30_2_DM260_Result_Data_64_bytes_1[71] := HwInputs.ST30_2_DM260_Result_Data_64_bytes_1[71];
END_FUNCTION
